(* IEC 61131-3 sources: brOscatLib/oscatNetw (part 2) *)

(* ---- DLOG_STORE_FILE_XML.st ---- *)
FUNCTION_BLOCK DLOG_STORE_FILE_XML
    (*http://www.oscat.de/images/OSCATBasic/oscat_basic333_en.pdf#page=46*)
    X.DTI := DTI; (* Datum / Zeit eintragen *)
    X.CLOCK_TRIG := DTI <> dti_last;
    dti_last := DTI;
    trig_auto := FALSE;
    IF X.CLOCK_TRIG THEN (* Impuls in jeder Sekunde *)
    	fn := DT_TO_STRF(DTI, 0, FILENAME, 0); (* automatische Dateinamen generierung *)
    	IF TRIG_T >= T#1000ms THEN (* automatischer Trigger *)
    		trig_auto := DT_TO_UDINT(DTI) MOD (TIME_TO_UDINT(TRIG_T) / UDINT#1000) = UDINT#0;
    	END_IF
    END_IF

    CASE step_1 OF

    00:	IF ENABLE THEN
    		aw_enable := AUTO_CLOSE >= T#5s;
    		wd_time := SEL(X.LOAD_TIME_MAX > T#0s, T#5ms,X.LOAD_TIME_MAX);
    		fn_last := fn; (* aktuellen Dateinnamen speichern *)
    		IF X.ID_MAX = USINT#0 THEN (* nur einmal nach Satellitenbausteinen scannen *)
    			X.ADD_COM := 01; (* ADD INFO *)
    			X.STORE_TYPE := BYTE#3; (* XML-Modus *)
    		END_IF
    		step_1 := 10;

    		(* ---------------- Debug-Message -----------------------*)
    		(*IF _debug_enable THEN
    			LOG_CL.NEW_MSG := 'FILE_XML1 - Start: File [~1], [~2]';
    			LOG_CL.PRINTF[1] := fn_last;
    			LOG_CL.PRINTF[2] := DT_TO_STRING(DTI);
    			LOG_MSG();
    		END_IF*)
    		(* -----------------------------------------------------------------*)

    	END_IF

    10:	X.UCB.D_STRING := fn_last;
    	IF fn_last = SAVE_DATA.FN_REM THEN
    		X.UCB.D_HEAD := WORD#16#F201; (* Filemode open + write *)
    		X.ADD_COM := 00;
    	ELSE
    		X.UCB.D_HEAD := WORD#16#F301; (* Filemode create + write *)
    		X.ADD_COM := 02; (* ADD HEADER *)
    	END_IF

    	X.UCB.D_MODE := 1; (* Dateinamen als String ablegen *)
    	UCB(DATA:=X.UCB); (* Daten eintragen *)
    	step_1 := 30;

    30:	(* LOG-Trigger verarbeiten *)
    	trig_tmp := (TRIG_M AND NOT trig_m_last) OR trig_auto OR X.ADD_DATA_REQ;

    	IF ENABLE = FALSE OR fn <> fn_last THEN (* ENABLE = 0 oder neuen Dateinamen -> Log Stop *)
    		trig_stored := trig_tmp; (* aktuellen Triggerpuls speichern *)
    		X.UCB.D_HEAD := WORD#16#EE00;
    		X.UCB.D_MODE := 1;
    		UCB(DATA:=X.UCB); (* Element schreiben *)
    		X.ADD_COM := 00;
    		step_1 := 00;

    		(* ---------------- Debug-Message -----------------------*)
    		(*IF _debug_enable THEN
    			LOG_CL.NEW_MSG := 'FILE_XML1 - Stop: [~2]';
    			LOG_CL.PRINTF[2] := DT_TO_STRING(DTI);
    			LOG_MSG();
    		END_IF*)
    		(* -----------------------------------------------------------------*)

    	ELSIF ENABLE THEN
    		IF trig_tmp OR trig_stored THEN (* manueller, automatischer oder externer Trigger *)
    			trig_stored := FALSE;
    			X.ADD_COM := 03; (* ADD DATA *)
    			SAVE_DATA.TRIG_CNT := SAVE_DATA.TRIG_CNT + UDINT#1;
    			SAVE_DATA.TRIG_CNT_TOTAL  := SAVE_DATA.TRIG_CNT_TOTAL + UDINT#1;
    			(* ---------------- Debug-Message -----------------------*)
    			(*IF _debug_enable THEN
    				LOG_CL.NEW_MSG := 'FILE_XML1 - Trig: [~2]';
    				LOG_CL.PRINTF[2] := DT_TO_STRING(DTI);
    				LOG_MSG();
    			END_IF*)
    			(* -----------------------------------------------------------------*)
    		ELSE
    			X.ADD_COM := 04;	(* ADD DATA REQ *)
    		END_IF
    	END_IF

    END_CASE
    X.ADD_DATA_REQ := FALSE; (* externe Anforderung rücksetzen *)

    (* ##################################### *)

    CASE step_2 OF

    00:	aw_ton(IN:= idx > 0 AND aw_enable , PT:= AUTO_CLOSE); (* AutoWrite Timer *)
    	IF aw_ton.Q THEN (* Zeitgesteuertes Datenschreiben *)
    		aw_aktiv := TRUE;
    		step_2 := 10; (* Daten schreiben *)
    		(* ---------------- Debug-Message -----------------------*)
    		(*IF _debug_enable THEN
    			LOG_CL.NEW_MSG := 'FILE_XML2 - AutoWrite: [~2]';
    			LOG_CL.PRINTF[2] := DT_TO_STRING(DTI);
    			LOG_MSG();
    		END_IF*)
    		(* -----------------------------------------------------------------*)

    	ELSE
    		wd_ton(IN:= FALSE, PT:= wd_time);
    		wd_ton(IN:= TRUE);
    		WHILE X.UCB.BUF_COUNT > 0 AND step_2 = 0 AND wd_ton.Q = FALSE DO

    			X.UCB.D_MODE := 10;
    			UCB(DATA:=X.UCB); (* Element lesen , aber noch nicht entfernen *)

    			IF X.UCB.D_HEAD > WORD#16#F000 THEN (* F301 oder F201 *)

    				str := '<?xml version="1.0" encoding="UTF-8"?><table>';

    				IF idx + LEN(str) < SIZEOF(PT.BUFFER) THEN (* Platz für Element vorhanden ? *)

    					FSD.MODE := WORD_TO_BYTE(SHR(SHL(X.UCB.D_HEAD,4),12)); (* 0X00 -> 000X = 3 create + write / 2 open + write *)
    					FSD.OFFSET := UDINT#0; (* Start bei Dateianfang *)
    					FSD.FILENAME := X.UCB.D_STRING; (* Dateiname *)
    					PT.SIZE := UINT#0;
    					SAVE_DATA.FN_REM := FSD.FILENAME; (* aktuellen Dateinamen remanent sichern *)

    					X.NEW_FILE := FSD.FILENAME;
    					X.NEW_FILE_SIZE := UDINT#0;
    					X.NEW_FILE_RTRIG := FALSE;
    					step_2 := 20;

    					(* Headerdaten schreiben *)
    					IF FSD.MODE = BYTE#3 THEN
    						SAVE_DATA.TRIG_CNT := UDINT#0; (* Datei neu anlegen -> dann zähler reset *)

    						_STRING_TO_BUFFER(str:=str, POS:=idx, PT:=ADR(PT.BUFFER), SIZE:=SIZEOF(PT.BUFFER));
    						idx := idx + LEN(str);
    						X.NEW_FILE_SIZE := total_bytes + INT_TO_UDINT(idx);
    					END_IF

    					X.UCB.D_MODE := 11;
    					UCB(DATA:=X.UCB); (* Element entfernen *)

    					(* ---------------- Debug-Message -----------------------*)
    					(*IF _debug_enable THEN
    						LOG_CL.NEW_MSG := 'FILE_XML2 - Create: Mode [~1] , [~2]';
    						LOG_CL.PRINTF[2] := DT_TO_STRING(DTI);
    						LOG_CL.PRINTF[1] := BYTE_TO_STRING(FSD.MODE);
    						LOG_MSG();
    					END_IF*)
    					(* -----------------------------------------------------------------*)
    				END_IF

    			ELSIF X.UCB.D_HEAD = WORD#16#EE00 THEN (* log_stop Command *)

    				str := '</table>';

    				IF idx + LEN(str) < SIZEOF(PT.BUFFER) THEN (* Platz für Element vorhanden ? *)

    					_STRING_TO_BUFFER(str:=str, POS:=idx, PT:=ADR(PT.BUFFER), SIZE:=SIZEOF(PT.BUFFER));
    					idx := idx + LEN(str);
    					log_stop := TRUE;
    					step_2 := 10; (* Daten schreiben *)

    					X.UCB.D_MODE := 11;
    					UCB(DATA:=X.UCB); (* Element entfernen *)

    				END_IF

    			ELSIF idx + LEN(X.UCB.D_STRING) + 120 < SIZEOF(PT.BUFFER) THEN (* Platz für Element vorhanden ? *)

    				(* ---------------- Debug-Message -----------------------*)
    				(*IF _debug_enable THEN
    					LOG_CL.NEW_MSG := 'FILE_XML2 - BUF: TXT [~1],Pos [~2], [~3]';
    					LOG_CL.PRINTF[1] := X.UCB.D_STRING;
    					LOG_CL.PRINTF[2] := INT_TO_STRING(idx);
    					LOG_CL.PRINTF[3] := DT_TO_STRING(DTI);
    					LOG_MSG();
    				END_IF*)
    				(* -----------------------------------------------------------------*)

    				IF log_state = USINT#0 THEN
    					str := '<row><entry>';
    				ELSE
    					str := '<entry>';
    				END_IF

    				_STRING_TO_BUFFER(str:=str, POS:=idx, PT:=ADR(PT.BUFFER), SIZE:=SIZEOF(PT.BUFFER));
    				idx := idx + LEN(str);
    				log_state := log_state + USINT#1;

    				_STRING_TO_BUFFER(str:=X.UCB.D_STRING, POS:=idx, PT:=ADR(PT.BUFFER), SIZE:=SIZEOF(PT.BUFFER));
    				idx := idx + LEN(X.UCB.D_STRING);

    				n := n + USINT#1;
    				IF n >= X.ID_MAX THEN
    					n := USINT#0;
    					str := '</entry></row>';
    					log_state := USINT#0;
    				ELSE
    					str := '</entry>';
    				END_IF
    				_STRING_TO_BUFFER(str:=str, POS:=idx, PT:=ADR(PT.BUFFER), SIZE:=SIZEOF(PT.BUFFER));
    				idx := idx + LEN(str);
    				X.NEW_FILE_SIZE := total_bytes + INT_TO_UDINT(idx);

    				X.UCB.D_MODE := 11;
    				UCB(DATA:=X.UCB); (* Element entfernen *)

    			ELSE (* kein Platz vorhanden *)
    				step_2 := 10; (* Daten schreiben *)
    			END_IF
    			wd_ton();
    		END_WHILE
    	END_IF

    10:	IF idx > 0 THEN (* Daten schreiben *)
    		FSD.MODE := BYTE#2; (* File_Open_Exist + File_Write *)
    		FSD.OFFSET := UDINT#4294967294; (* 16#FFFF_FFFE ->Spezialcode: Daten automatisch an Dateiende anhängen *)
    		PT.SIZE := INT_TO_UINT(idx); (* Datenlänge eintragen *)
    		idx := 0;
    		(* ---------------- Debug-Message -----------------------*)
    		(*IF _debug_enable THEN
    			LOG_CL.NEW_MSG := 'FILE_XML2 - WriteData: Mode [~3] Size [~1] , [~2]';
    			LOG_CL.PRINTF[1] := UINT_TO_STRING(PT.SIZE);
    			LOG_CL.PRINTF[2] := DT_TO_STRING(DTI);
    			LOG_CL.PRINTF[3] := BYTE_TO_STRING(FSD.MODE);
    			LOG_MSG();
    		END_IF*)
    		(* -----------------------------------------------------------------*)
    	END_IF
    	step_2 := 20;

    20:	IF FSD.MODE = BYTE#0 THEN
    		total_bytes := FSD.FILE_SIZE;
    		X.NEW_FILE_SIZE := total_bytes + INT_TO_UDINT(idx);
    		IF log_stop OR aw_aktiv THEN
    			aw_aktiv := FALSE;
    			FSD.MODE := BYTE#5; (* Datei schliessen *)
    			(* ---------------- Debug-Message -----------------------*)
    			(*IF _debug_enable THEN
    				LOG_CL.NEW_MSG := 'FILE_XML2 - Close: [~2]';
    				LOG_CL.PRINTF[2] := DT_TO_STRING(DTI);
    				LOG_MSG();
    			END_IF*)
    			(* -----------------------------------------------------------------*)
    		END_IF
    		step_2 := 30;
    	END_IF

    30:	IF FSD.MODE = BYTE#0 THEN (* Datei schliessen beendet *)
    		IF log_stop THEN
    			X.NEW_FILE_RTRIG := TRUE;
    			log_stop := FALSE;
    			SAVE_DATA.FN_REM := ''; (* remanenten Dateinamen löschen *)
    		END_IF
    		step_2 := 00;
    	END_IF

    END_CASE

    FS(FSD:=FSD,PT:=PT); (* FILE_SERVER *)

    (* Fehlerauswertung *)
    IF FSD.ERROR <> BYTE#0 THEN
    	ERROR_C := BYTE_TO_DWORD(FSD.ERROR);
    	ERROR_T := BYTE#1;
    ELSIF X.UCB.BUF_DATA_LOST > UDINT#0 THEN
    	ERROR_C := DWORD#2; (* Fehler: Bufferüberlauf - Datenmenge reduzieren *)
    	ERROR_T := BYTE#6; 	(* Type: Buffer *)
    ELSIF X.UCB.BUF_USED_MAX > USINT#90 THEN
    	ERROR_C := DWORD#1; (* Warnung: Buffer auslastung > 90% *)
    	ERROR_T := BYTE#6;	(* Type: Buffer *)
    ELSE
    	ERROR_C := DWORD#0;
    	ERROR_T := BYTE#0;
    END_IF

    trig_m_last := TRIG_M;

    (* revision history
    ks	25. july. 2011	rev 1.0
    	original version

    ks	16. apr. 2012	rev 1.1
    	neuer überarbeiteter Code für automatisches File-open/close

    ks	8. mar. 2016	rev 1.2
    	nur einmal nach satellitenbausteinen scannen

    ks	21. mar. 2016	rev 1.3
    	prüfung auf freien bufferplatz hinzugefügt
    	fehlermeldungen hinzugefügt

    *)
END_FUNCTION_BLOCK

(* ---- DLOG_STORE_MYSQL.st ---- *)
FUNCTION_BLOCK DLOG_STORE_MYSQL
    (*http://www.oscat.de/images/OSCATBasic/oscat_basic333_en.pdf#page=46*)
    X.DTI := DTI; (* Datum / Zeit eintragen *)
    X.CLOCK_TRIG := DTI <> dti_last;
    dti_last := DTI;
    trig_auto := FALSE;
    IF X.CLOCK_TRIG THEN (* Impuls in jeder Sekunde *)
    	del_start := DT_TO_UDINT(DTI) - del_dt > AUTO_DELETE AND AUTO_DELETE > UDINT#0;
    	IF TRIG_T >= T#1000ms THEN (* automatischer Trigger *)
    		trig_auto := DT_TO_UDINT(DTI) MOD (TIME_TO_UDINT(TRIG_T) / UDINT#1000) = UDINT#0;
    	END_IF
    END_IF
    X.ADD_COM := 00;

    CASE step OF

    00:	IF ENABLE AND enable_last = FALSE THEN
    		y.SQL_URL := URL;
    		y.TIMEOUT := TIMEOUT;
    		y.DNS_IP4 := DNS_IP4;
    		y.SQL_CON := TRUE;

    		X.UCB.D_MODE := 99; (* Buffer reset - Alles löschen *)
    		UCB(DATA:=X.UCB);

    		IF X.ID_MAX = USINT#0 THEN (* nur einmal nach Satellitenbausteinen scannen *)
    			X.ADD_COM := 01; (* ADD INFO *)
    			X.STORE_TYPE := BYTE#5; (* MySQL-Modus *)
    		END_IF

    		step := 05;
    	END_IF

    05:	X.ADD_COM := 02; (* ADD HEADER *)
    	step := 10;

    10:	IF SQL_INFO.SQL_CONNECTED THEN
    		sql_command := BYTE#3; (* CREATE DATABASE IF NOT EXISTS `DB_NAME` *)
    		snd_text :=  CONCAT('CREATE DATABASE IF NOT EXISTS `' ,DB_NAME);
    		snd_text :=  CONCAT(snd_text, '`');
    		next_step := 20;
    	END_IF

    20:	sql_command := BYTE#2; (* 0x02 COM_INIT_DB mysql_select_db *)
    	snd_text := DB_NAME;
    	next_step := 30;

    30:	(* CREATE TABLE IF NOT EXISTS TB_NAME (Timestamp TIMESTAMP NULL DEFAULT CURRENT_TIMESTAMP, n1,n2) *)
    	sql_command := BYTE#0;
    	idx := 5;
    	n := USINT#0;
    	WHILE sql_command = BYTE#0 DO
    		IF n = USINT#0 THEN
    			snd_text := CONCAT('CREATE TABLE IF NOT EXISTS `', TB_NAME);
    			snd_text := CONCAT(snd_text,'` (`ID` BIGINT NOT NULL AUTO_INCREMENT PRIMARY KEY ,');
    			snd_text := CONCAT(snd_text,' store_timestamp TIMESTAMP NULL DEFAULT CURRENT_TIMESTAMP');
    		ELSIF n <= X.ID_MAX THEN
    			X.UCB.D_MODE := 12; (* Element lesen und löschen *)
    			UCB(DATA:=X.UCB);
    			snd_text := CONCAT(', `',X.UCB.D_STRING);
    			CASE WORD_TO_INT(SHR(X.UCB.D_HEAD,8)) OF
    			02:	snd_text := CONCAT(snd_text, '` FLOAT'); (* REAL *)
    			06:	snd_text := CONCAT(snd_text, '` BOOL'); (* BOOL *)
    			08:	snd_text := CONCAT(snd_text, '` INT'); (* DINT *)
    			13:	snd_text := CONCAT(snd_text, '` DATETIME'); (* DT *)
    			ELSE
    				snd_text := CONCAT(snd_text, '` VARCHAR(80)'); (* STRING(80) *)
    			END_CASE
    		ELSE
    			snd_text := ')';
    			sql_command := BYTE#3;
    			snd_size := idx + LEN(snd_text);
    			next_step := 40;
    		END_IF
    		_STRING_TO_BUFFER(str:=snd_text,pos:=idx,pt:=ADR(y.S_BUF.BUFFER),size:=SIZEOF(y.S_BUF.BUFFER)); (* String in puffer kopieren *)
    		idx := idx + LEN(snd_text);
    		n := n + USINT#1;

    		(*####################  DEBUG-MESSAGE  ###################################*)
    		(*IF _debug_enable THEN
    			LOG_CL.NEW_MSG := 'dlog_mysql: create >~1<';
    			LOG_CL.PRINTF[1] := snd_text;
    			LOG_MSG();
    		END_IF*)
    		(*########################################################################*)
    	END_WHILE

    40:	IF del_start THEN
    		del_start := FALSE;
    		sql_command := BYTE#3; (* DELETE FROM `TB_NAME` WHERE TIMESTAMPDIFF(SECOND, Timestamp, NOW()) > xxx *)
    		snd_text := CONCAT('DELETE FROM `', TB_NAME);
    		snd_text := CONCAT(snd_text, '` WHERE TIMESTAMPDIFF(SECOND, store_timestamp, NOW()) > ');
    		snd_text := CONCAT(snd_text, UDINT_TO_STRING(AUTO_DELETE));
    		next_step := 40;
    		del_dt := DT_TO_UDINT(DTI);
    		(*####################  DEBUG-MESSAGE  ###################################*)
    		(*IF _debug_enable THEN
    			LOG_CL.NEW_MSG := 'dlog_mysql: # delete time:~1 >~2<';
    			LOG_CL.PRINTF[1] := UDINT_TO_STRING(AUTO_DELETE);
    			LOG_CL.PRINTF[2] := snd_text;
    			LOG_MSG();
    		END_IF*)
    		(*########################################################################*)

             (* INSERT INTO `TB_NAME` VALUES (CURRENT_TIMESTAMP,  "n1","n2") *)
    	ELSIF X.UCB.BUF_COUNT >= USINT_TO_INT(X.ID_MAX) AND step > 0 THEN (* Neue Datenreihe(n) vorhanden *)
    		idx := 5;
    		n := USINT#0;
    		sql_command := BYTE#0;
    		WHILE sql_command = BYTE#0 DO
    			IF n = USINT#0 THEN
    				snd_text := CONCAT('INSERT INTO `', TB_NAME);
    				snd_text := CONCAT(snd_text,'` VALUES (NULL, CURRENT_TIMESTAMP');
    			ELSIF n <= X.ID_MAX THEN
    				X.UCB.D_MODE := 12; (* Element lesen und löschen *)
    				UCB(DATA:=X.UCB);
    				snd_text := CONCAT(', "',X.UCB.D_STRING);
    				snd_text := CONCAT(snd_text, '"');
    			ELSE
    				snd_text := ')';
    				sql_command := BYTE#3;
    				snd_size := idx + LEN(snd_text);
    				next_step := 40;
    			END_IF
    			_STRING_TO_BUFFER(str:=snd_text,pos:=idx,pt:=ADR(y.S_BUF.BUFFER),size:=SIZEOF(y.S_BUF.BUFFER)); (* String in puffer kopieren *)
    			idx := idx + LEN(snd_text);
    			n := n + USINT#1;

    			(*####################  DEBUG-MESSAGE  ###################################*)
    			(*IF _debug_enable THEN
    				LOG_CL.NEW_MSG := 'dlog_mysql: insert >~1<';
    				LOG_CL.PRINTF[1] := snd_text;
    				LOG_MSG();
    			END_IF*)
    			(*########################################################################*)
    		END_WHILE
    	END_IF

    	IF ENABLE THEN 	(* LOG-Trigger verarbeiten *)
    		trig_tmp := (TRIG_M AND NOT trig_m_last) OR trig_auto OR X.ADD_DATA_REQ;

    		IF trig_tmp THEN (* manueller, automatischer oder externer Trigger *)
    			X.ADD_COM := 03; (* ADD DATA *)
    			(* ---------------- Debug-Message -----------------------*)
    			(*IF _debug_enable THEN
    				LOG_CL.NEW_MSG := 'dlog_mysql: Trigger: DATE [~2]';
    				LOG_CL.PRINTF[2] := DT_TO_STRING(DTI);
    				LOG_MSG();
    			END_IF*)
    			(* -----------------------------------------------------------------*)
    		ELSE
    			X.ADD_COM := 04;	(* ADD DATA REQ *)
    		END_IF
    	ELSE
    		y.SQL_CON := FALSE; (* MySQL Verbindung beenden *)
    		step := 0;
    	END_IF
    	X.ADD_DATA_REQ := FALSE;

    (* ~~~~~~~~~~~~~~~~~~~~~~ *)

    199:IF y.SQL_RCV_STATE = BYTE#1 THEN (* OK *)
    		step := next_step;
    	ELSIF y.SQL_RCV_STATE = BYTE#2 THEN  (* FEHLER *)
    		step := 0;
    	END_IF

    END_CASE

    (* ########################## *)
    (* SQL-Kommando ausführen *)
    IF sql_command > BYTE#0 THEN

    	IF snd_size > 0 THEN
    		y.S_BUF.SIZE := INT_TO_UINT(snd_size);
    		snd_size := 0;
    	ELSE
    		_STRING_TO_BUFFER(str:=snd_text,pos:=5,pt:=ADR(y.S_BUF.BUFFER),size:=SIZEOF(y.S_BUF.BUFFER)); (* String in puffer kopieren *)
    		y.S_BUF.SIZE := INT_TO_UINT(5 + LEN(snd_text));
    		snd_text := '';
    	END_IF

    	IF y.S_BUF.SIZE > SIZEOF(y.S_BUF.BUFFER) THEN (* buffer überlauf erkannt -> Abbruch *)
    		y.S_BUF.SIZE := 0;
    		sql_command := BYTE#0;
    		y.SQL_CON := FALSE; (* MySQL Verbindung beenden *)
    		step := 999; (* Dummy-Schritt *)
    	ELSE

    		i2 := UINT_TO_INT(y.S_BUF.SIZE) - 1; (* alle " zeichen mit ' ersetzen *)
    		FOR i1 := 5 TO i2 DO
    			IF y.S_BUF.BUFFER[i1] = BYTE#34 THEN
    				y.S_BUF.BUFFER[i1] := BYTE#39;
    			END_IF
    		END_FOR

    		y.S_BUF.BUFFER[4] := sql_command;
    		y.SQL_PACKET_NO := BYTE#255;
    		sql_command := BYTE#0;
    		step := 199;
    	END_IF
    END_IF

    (* ########################## *)

    MYSQL_CONTROL(COM:= y, INFO:=SQL_INFO);

    (* Fehlerauswertung *)
    IF step = 999 THEN	(* Buffer überlauf *)
    	ERROR_C := DWORD#3; (* Netzwerkbuffer überlauf *)
    	ERROR_T := BYTE#6; 	(* Type: Buffer *)
    ELSIF y.ERROR_T > BYTE#0 THEN	(* SQL Error *)
    	ERROR_C := y.ERROR_C;
    	ERROR_T := y.ERROR_T;
    	step := 0;
    ELSIF X.UCB.BUF_DATA_LOST > UDINT#0 THEN
    	ERROR_C := DWORD#2; (* Fehler: Bufferüberlauf - Datenmenge reduzieren *)
    	ERROR_T := BYTE#6; 	(* Type: Buffer *)
    ELSIF X.UCB.BUF_USED_MAX > USINT#90 THEN
    	ERROR_C := DWORD#1; (* Warnung: Buffer auslastung > 90% *)
    	ERROR_T := BYTE#6;	(* Type: Buffer *)
    ELSE
    	ERROR_C := DWORD#0;
    	ERROR_T := BYTE#0;
    END_IF

    (* ########################## *)

    trig_m_last := TRIG_M;
    enable_last := ENABLE;
    run := step > 0;

    (* revision history
    ks	20. apr. 2012	rev 1.0
    	original version

    ks	17. jan. 2014	rev 1.1
    	DELTA Error

    ks	8. mar. 2016	rev 1.2
    	nur einmal nach satellitenbausteinen scannen

    ks	21. mar. 2016	rev 1.3
    	prüfung auf bufferüberlauf und fehlermeldungen hinzugefügt

    *)
END_FUNCTION_BLOCK

(* ---- DLOG_STORE_RRD.st ---- *)
FUNCTION_BLOCK DLOG_STORE_RRD
    (*http://www.oscat.de/images/OSCATNetwork/oscat_netlib121_en.pdf#page=54*)
    X.DTI := DTI; (* Datum / Zeit eintragen *)
    X.CLOCK_TRIG := DTI <> dti_last;
    dti_last := DTI;
    trig_auto := FALSE;
    IF X.CLOCK_TRIG THEN (* Impuls in jeder Sekunde *)
    	IF TRIG_T >= T#1000ms THEN (* automatischer Trigger *)
    		trig_auto := DT_TO_UDINT(DTI) MOD (TIME_TO_UDINT(TRIG_T) / UDINT#1000) = UDINT#0;
    	END_IF
    END_IF

    CASE step_1 OF

    00:	IF ENABLE THEN
    		IF X.ID_MAX = USINT#0 THEN (* nur einmal nach Satellitenbausteinen scannen *)
    			X.ADD_COM := 01; (* ADD INFO *)
    			X.STORE_TYPE := BYTE#1; (* RRD-Modus *)
    		END_IF

    		ERROR_T := BYTE#0;
    		ERROR_C := DWORD#0;

    		X.UCB.D_MODE := 99;
    		UCB(DATA:=X.UCB); (* Buffer löschen *)

    		URL_DATA:=STRING_TO_URL(STR:=URL,DEFAULT_PROTOCOL:='',DEFAULT_PATH:=''); (* URL zerlegen *)
    		sep_char := CHR_TO_STRING(SEP);
    		url_query := URL_DATA.QUERY;
    		step_1 := 30;

    		(* ---------------- Debug-Message -----------------------*)
    		(*IF _debug_enable THEN
    			LOG_CL.NEW_MSG := 'FILE_RRD1 - Start: DATE [~2]';
    			LOG_CL.PRINTF[2] := DT_TO_STRING(DTI);
    			LOG_MSG();
    		END_IF*)
    		(* -----------------------------------------------------------------*)

    	END_IF

    30:	(* LOG-Trigger verarbeiten *)
    	trig_tmp := (TRIG_M AND NOT trig_m_last) OR trig_auto OR X.ADD_DATA_REQ;

    	IF ENABLE = FALSE THEN (* ENABLE = 0 -> Log Stop *)
    		X.ADD_COM := 00;
    		step_1 := 00;

    		(* ---------------- Debug-Message -----------------------*)
    		(*IF _debug_enable THEN
    			LOG_CL.NEW_MSG := 'FILE_RRD1 - Stop: DATE [~2]';
    			LOG_CL.PRINTF[2] := DT_TO_STRING(DTI);
    			LOG_MSG();
    		END_IF*)
    		(* -----------------------------------------------------------------*)

    	ELSIF ENABLE THEN
    		IF trig_tmp OR trig_stored THEN (* manueller, automatischer oder externer Trigger *)
    			trig_stored := FALSE;
    			X.ADD_COM := 03; (* ADD DATA *)
    			(* ---------------- Debug-Message -----------------------*)
    			(*IF _debug_enable THEN
    				LOG_CL.NEW_MSG := 'FILE_RRD1 - Trig: DATE [~2]';
    				LOG_CL.PRINTF[2] := DT_TO_STRING(DTI);
    				LOG_MSG();
    			END_IF*)
    			(* -----------------------------------------------------------------*)
    		ELSE
    			X.ADD_COM := 04;	(* ADD DATA REQ *)
    		END_IF
    	END_IF

    END_CASE
    X.ADD_DATA_REQ := FALSE; (* externe Anforderung rücksetzen *)

    (* ##################################### *)

    CASE step_2 OF

    00:	IF X.UCB.BUF_DATA_LOST > UDINT#0 THEN
    		ERROR_C := DWORD#2; (* Fehler: Bufferüberlauf - Datenmenge reduzieren *)
    		ERROR_T := BYTE#6; 	(* Type: Buffer *)
    		step_2 := 100;
    	ELSIF X.UCB.BUF_USED_MAX > USINT#90 THEN
    		ERROR_C := DWORD#1; (* Warnung: Buffer auslastung > 90% *)
    		ERROR_T := BYTE#6;	(* Type: Buffer *)
    	END_IF

    	IF X.UCB.BUF_COUNT >= USINT_TO_INT(X.ID_MAX) THEN (* genug Einträge vorhanden *)
    		URL_DATA.QUERY := url_query; (* original Query wiederherstellen *)
    		n := 1;
    		WHILE n <= USINT_TO_INT(X.ID_MAX) DO
    			X.UCB.D_MODE := 12; (* Element lesen und löschen *)
    			UCB(DATA:=X.UCB);
    			IF n < USINT_TO_INT(X.ID_MAX) THEN (* Trennzeichen hinzufügen *)
    				X.UCB.D_STRING := CONCAT(X.UCB.D_STRING,sep_char);
    			END_IF
    			IF LEN(X.UCB.D_STRING) + LEN(URL_DATA.QUERY) <= STRING_LENGTH THEN
    				URL_DATA.QUERY := CONCAT(URL_DATA.QUERY,X.UCB.D_STRING); (* Query mit LOG-Daten ergänzen *)
    				step_2 := 40;
    			ELSE
    				ERROR_T := BYTE#4; (* LOG-Daten können nicht in URL gepackt werden *)
    				ERROR_C := DWORD#1;
    				step_2 := 100;
    			END_IF
    			n := n + 1;
    		END_WHILE;
    	END_IF

    40:	IF DNS_CLIENT.DONE THEN
    		step_2 := 60;
    	ELSIF (DNS_CLIENT.ERROR > DWORD#0) THEN
    		ERROR_C := DNS_CLIENT.ERROR; (* Fehlerbehandlung *)
    		ERROR_T := BYTE#1;
    		step_2 := 100;
    	END_IF

    60:	IF HTTP_GET.DONE THEN
    		n := UINT_TO_INT(HTTP_GET.BODY_START);
    		IF R_BUF.BUFFER[n] <> BYTE#48 THEN (* ASCII '0' *)
    			ERROR_C := DWORD#1;
    			ERROR_T := BYTE#3;
    		END_IF
    		step_2 := 100;

    	ELSIF HTTP_GET.ERROR > DWORD#0 THEN (* Fehlerbehandlung *)
    		ERROR_C := HTTP_GET.ERROR;
    		ERROR_T := BYTE#2;
    		step_2 := 100;
    	END_IF

    100:	IF (NOT HTTP_GET.DONE) THEN (* UNLOCK HTTP DATA *)
    		step_2 := SEL(ERROR_T = BYTE#0, 120,0);
    	END_IF

    120:	IF NOT ENABLE THEN
    		step_2 := 0;
    	END_IF

    END_CASE

    HTTP_GET(IP_C:=IP_C,S_BUF:=S_BUF,R_BUF:=R_BUF,IP4:=DNS_CLIENT.IP4,GET:=step_2=60,MODE:=2,UNLOCK_BUF:=step_2=100,URL_DATA:=URL_DATA); (* HTTP_GET *)
    DNS_CLIENT(IP_C:=IP_C, S_BUF:=S_BUF, R_BUF:=R_BUF, DOMAIN:=URL_DATA.DOMAIN, IP4_DNS:= DNS_IP4, ACTIVATE:=step_2=40); (* DNS-Client *)
    IPC(IP:= 0, PORT:= 0 , TIME_OUT:= TIMEOUT, IP_C:= IP_C, S_BUF:= S_BUF, R_BUF:= R_BUF); (* IP_CONTROL *)

    trig_m_last := TRIG_M;

    (* revision history
    ks	01. jan. 2011	rev 1.0
    	original version

    ks	13. may. 2011	rev 1.1
    	ADD_DATA_REQ hinzugefügt

    ks	26. july. 2011	rev 1.2
    	code optimierung D_MODE 12 und bessere fehlerauswertung

    ks	16. apr. 2012	rev 1.3
    	neuer überarbeiteter Code

    ks	21. mar. 2016	rev 1.4
    	nur einmal nach satellitenbausteinen scannen und fehlermeldungen hinzugefügt

    *)
END_FUNCTION_BLOCK

(* ---- DLOG_STRING.st ---- *)
FUNCTION_BLOCK DLOG_STRING
    (*http://www.oscat.de/images/OSCATNetwork/oscat_netlib121_en.pdf#page=52*)
    CASE X.ADD_COM OF

    01:	(* ADD INFO *)
    	X.ID_MAX := X.ID_MAX + USINT#1;
    	id := WORD#16#0101; (* Quelltype STRING , Zieltype STRING *)
    02:	(* ADD HEADER *)
    	X.UCB.D_STRING := COLUMN;
    	X.UCB.D_HEAD := id;
    	X.UCB.D_MODE := 1;
    	UCB(DATA:=X.UCB); (* Daten eintragen *)
    03:	(* ADD DATA *)
    	X.UCB.D_STRING := str_last;
    	X.UCB.D_HEAD := id;
    	X.UCB.D_MODE := 1;
    	UCB(DATA:=X.UCB); (* Daten eintragen *)
    END_CASE
    str_last := STR;

    (* revision history
    ks	01. jan. 2011	rev 1.0
    	original version

    ks	17. may. 2011	rev 1.1
    	COLUMN STRING(40)

    ks	25. july.   2011	rev 1.2
    	neue head information

    ks	19. apr.   2012	rev 1.3
    	code neu überarbeitet
    *)
END_FUNCTION_BLOCK

(* ---- DNS_CLIENT.st ---- *)
FUNCTION_BLOCK DNS_CLIENT
    (*http://www.oscat.de/images/OSCATNetwork/oscat_netlib121_en.pdf#page=89*)
    (* DOMAIN Name System (query) *)

    CASE state OF

    00:	IF ACTIVATE AND NOT activate_last THEN (* auf positive Flanke GET warten *)
    		DONE := FALSE;
    		ERROR := DWORD#0;
    		state := 5;
    	END_IF

    05:	IP4 := IP4_DECODE(str:=DOMAIN); (* prüfe ob DOMAIN schon eine IP4-Adresse ist *)
    	IF IP4 > DWORD#00 THEN
    		DONE := TRUE;
    		state := 0;
            		(*####################  DEBUG-MESSAGE  ###################################*)
            		(*IF _debug_enable THEN
                		LOG_CL.NEW_MSG := 'DNS: S05 IP4 ~1';
                		LOG_CL.PRINTF[1]  := DOMAIN;
                		LOG_MSG();
            		END_IF*)
            		(*########################################################################*)
    	ELSE
    		ip_state := BYTE#1;
    		ttl_last := DWORD#0;
    		domain_copy := DOMAIN; (* DOMAIN String sichern *)
    		state := 10;
            		(*####################  DEBUG-MESSAGE  ###################################*)
            		(*IF _debug_enable THEN
                		LOG_CL.NEW_MSG := 'DNS: S05 START';
                		LOG_MSG();
            		END_IF*)
            		(*########################################################################*)
    	END_IF

    10:	IF ip_state = BYTE#3 THEN (* Bei IP_Control anmelden *)
    		url_length := LEN(domain_copy);
    		char_count := 17 + url_length; (* sendebuffer initialisieren *)
    		FOR i := 0 TO char_count DO
    			S_BUF.BUFFER[i] := BYTE#00;
    		END_FOR
    		tid := UINT_TO_BYTE(BYTE_TO_UINT(tid) + UINT#1);
    		S_BUF.BUFFER[01] := tid; (* Transaction ID lowbyte *)
    		S_BUF.BUFFER[02] := BYTE#16#01; (* Flags: highbyte *)
    		S_BUF.BUFFER[05] := BYTE#16#01; (* Questions: lowbyte *)
    		i := url_length + 12;	(* den servernamen von hinten nach vorne bearbeiten *)
    		char_count := 0;
    		WHILE i > 12 DO
    			char := CODE(STR:=domain_copy,POS:=i - 12);
    			IF char = BYTE#46 THEN (* prüfe auf haupt/sub domänen namens-teiler "." *)
    				S_BUF.BUFFER[i] := INT_TO_BYTE(char_count); (* anstelle des teilers "." wird die länge des erkannten haupt/sub domänennames eingetragen *)
    				char_count := 0;
    			ELSE
    				S_BUF.BUFFER[i] := char; (* char in buffer eintragen *)
    				char_count := char_count + 1; (* anzahl char zählen *)
    			END_IF
    			i := i - 1;
    		END_WHILE
    		S_BUF.BUFFER[i] := INT_TO_BYTE(char_count); (* längenangabe des ganz linken (ersten) domänennamens eintragen *)
    		i := url_length + 15; (* position hinter dem servernamen *)
    		S_BUF.BUFFER[i] := BYTE#01; (* Type: A Hostaddress lowbyte *)
    		i := i + 2;
    		S_BUF.BUFFER[i] := BYTE#01; (* Class: IN lowbyte *)
    		i := i + 1;
    		(* IP Datenverkehr einrichten *)
    		IP_C.C_PORT := WORD#53; (* Portnummer eintragen *)
    		IP_C.C_IP := IP4_DNS; (* IP eintragen *)
    		IP_C.C_MODE := BYTE#1; (* Mode: UDP+AKTIV+PORT+IP *)
    		IP_C.C_ENABLE := TRUE; (* Verbindungsaufbau freigeben *)
    		IP_C.TIME_RESET := TRUE; (* Zeitueberwachung rücksetzen *)
    		IP_C.R_OBSERVE  := TRUE; (* Datenempfang ueberwachen *)
    		S_BUF.SIZE := INT_TO_UINT(i); (* sendelänge eintragen *)
    		R_BUF.SIZE := UINT#0; (* Empfangslänge rücksetzen *)
    		state := 30;

            		(*####################  DEBUG-MESSAGE  ###################################*)
            		(*IF _debug_enable THEN
                		LOG_CL.NEW_MSG := 'DNS: S10 SEND';
                		LOG_MSG();
            		END_IF*)
            		(*########################################################################*)
    	END_IF

    30:	IF IP_C.ERROR <> DWORD#00 THEN
    		ERROR := IP_C.ERROR;
    		state := 99;
            		(*####################  DEBUG-MESSAGE  ###################################*)
            		(*IF _debug_enable THEN
                		LOG_CL.NEW_MSG := 'DNS: S30 ERROR ~1';
                		LOG_CL.PRINTF[1]  := DWORD_TO_STRING(ERROR);
                		LOG_MSG();
            		END_IF*)
            		(*########################################################################*)

    	ELSIF (S_BUF.SIZE = UINT#0) AND (tid = R_BUF.BUFFER[1]) AND (R_BUF.SIZE >= INT_TO_UINT(34 + url_length)) THEN	(* prüfe ob antwort telegramm die richtige Transaction-ID und mindestlänge hat *)
    		ERROR := BYTE_TO_DWORD(R_BUF.BUFFER[3] AND BYTE#2#0000_1111); (* prüfe Return code der Flags. 4 bits *)
    		IF ERROR = DWORD#00 THEN
    			anc := R_BUF.BUFFER[7]; (* Anzahl der Answer-RR *)
    			IP_C.R_OBSERVE := FALSE; (* Datenempfang ueberwachen *)
    			state := 40;
    		ELSE
    			state := 99;
    		END_IF
    	END_IF

    40:	IF anc > 0 THEN
    		anc := anc - 1;
    		WHILE i < R_BUF.SIZE DO
    			x := R_BUF.BUFFER[i];
    			IF rr_stop = FALSE THEN
    				IF x > BYTE#63 THEN (* zeiger auf namen *)
    					i := i + 1;
    					rr_stop := TRUE;
    				ELSIF x= BYTE#0 THEN (* namens ende *)
    					rr_stop := TRUE;
    				ELSE
    					i := i + x; (* namen *)
    				END_IF
    				i := i + 1;
    			ELSE
    				rr_stop := FALSE;
    				IF R_BUF.BUFFER[i+1] = BYTE#1 AND R_BUF.BUFFER[i+3] = BYTE#1 THEN (* Type A / Class IN *)
    					i := i + 4;
    					ttl_tmp := DWORD_OF_BYTE(R_BUF.BUFFER[i],R_BUF.BUFFER[i+1],R_BUF.BUFFER[i+2],R_BUF.BUFFER[i+3]); (* Time to live *)
    					i := i + 6;
    					IF ttl_tmp >= ttl_last THEN (* TTL ist länger *)
    						ttl_last := ttl_tmp;
    						IP4 := DWORD_OF_BYTE(R_BUF.BUFFER[i],R_BUF.BUFFER[i+1],R_BUF.BUFFER[i+2],R_BUF.BUFFER[i+3]); (* IP-Adresse *)
    					END_IF
    					i := i + 4;
    				ELSE
    					i := i + 9;
    					i := i + R_BUF.BUFFER[i] + 1; (* offset zu nächsten Block *)
    				END_IF
    				EXIT;
    			END_IF
    		END_WHILE
    	ELSE
    		IF IP4 > DWORD#0 THEN (* gültige RR mit IP gefunden *)
    			DONE := TRUE;
                		(*####################  DEBUG-MESSAGE  ###################################*)
                		(*IF _debug_enable THEN
                    			LOG_CL.NEW_MSG := 'DNS: S40 OK';
                    			LOG_MSG();
                		END_IF*)
                		(*########################################################################*)
    		ELSE
    			ERROR := DWORD#255; (* Daten fehlerhaft - keine IP-Adresse vorhanden *)
    		END_IF
    		state := 99;
    	END_IF

    99:	R_BUF.SIZE := UINT#0; (* Empfangslänge rücksetzen *)
    	ip_state := BYTE#4; (* Abmelden *)
    	state := 00;

    END_CASE

    activate_last := ACTIVATE; (* letzten Status sichern zur Flankenerkennung *)
    IP_FIFO(FIFO:=IP_C.FIFO,state:=ip_state,ID:=ip_id); (* IP_FIFO *)

    (* revision history

    ks	18. oct. 2008	rev 1.0
    	original version

    ks	20. oct. 2009	rev 1.1
    	unbenutzten code entfernt, all buffer base 0

    ks	20. dec. 2010	rev 1.2
    	parsing nach rfc1305

    ks	26. jul. 2011	rev 1.3
    	verbesserte ip-auswertung , neue fehlermeldung
    *)

    (*----------------------------------------------------------------------------------------------------------------*)
    (* Flags: 0x0100 (Standard query)                                                                                            *)
    (* 0... .... .... .... = Response: Message is a query                                                                   *)
    (* .000 0... ....  = Opcode: Standard query (0)                                                                          *)
    (* .... ..0. .... .... = Truncated: Message is not truncated                                                          *)
    (* .... ...1 .... .... = Recursion desired: Do query recursively                                                    *)
    (* .... .... .0.. .... = Z: reserved (0)                                                                                                  *)
    (* .... .... ...0 .... = Non-authenticated data OK: Non-authenticated data is unacceptable *)
    (*-----------------------------------------------------------------------------------------------------------------*)

    (*      0  1  2  3  4  5  6  7  8  9  0  1  2  3  4  5  *)
    (*    +--+--+--+--+--+--+--+--+--+--+--+--+--+--+--+--+ *)
    (*    |                      ID                       | idx: 0/1   *)
    (*    +--+--+--+--+--+--+--+--+--+--+--+--+--+--+--+--+ *)
    (*    |QR|   Opcode  |AA|TC|RD|RA|   Z    |   RCODE   | idx: 2/3   *)
    (*    +--+--+--+--+--+--+--+--+--+--+--+--+--+--+--+--+ *)
    (*    |                    QDCOUNT                    | idx: 4/5   *)
    (*    +--+--+--+--+--+--+--+--+--+--+--+--+--+--+--+--+ *)
    (*    |                    ANCOUNT                    | idx: 6/7   *)
    (*    +--+--+--+--+--+--+--+--+--+--+--+--+--+--+--+--+ *)
    (*    |                    NSCOUNT                    | idx: 8/9   *)
    (*    +--+--+--+--+--+--+--+--+--+--+--+--+--+--+--+--+ *)
    (*    |                    ARCOUNT                    | idx: 10/11 *)
    (*    +--+--+--+--+--+--+--+--+--+--+--+--+--+--+--+--+ *)

    (*
    Errorcodes  Description	References
    000	No ERROR. 		 	The request completed successfully.
    001	Format ERROR. 		The name server was unable to interpret the query.
    002	Server failure.  	The name server was unable to process this query due to a problem with the name server.
    003	Name ERROR. 	 	Meaningful only for responses from an authoritative name server, this code signifies that the DOMAIN name referenced in the query does not exist.
    004	Not Implemented. 	The name server does not support the requested kind of query.
    005	Refused. 			The name server refuses to perform the specified operation for policy reasons.
      						 For example, a name server may not wish to provide the information to the particular requester, or a name server may not wish to perform a particular operation (e.g., zone transfer) for particular data.
    006	YXDomain.			Name Exists when it should not.
    007	YXRRSet. RR			Set Exists when it should not.
    008	NXRRSet. RR			Set that should exist does not.
    009	NotAuth.			Server Not Authoritative for zone.
    010	NotZone,			Name not contained in zone.
    255	Timeout				No Response

    beispiel einer DNS Request von google.at
    ein request mit 3 Answer-Blocks

    DOMAIN Name System (response)
    [Request In: 3]
    [Time: 0.027533000 seconds]
    Transaction ID: 0x5e1a
    Flags: 0x8180 (Standard query response, No ERROR)
    1... .... .... .... = Response: Message is a response
    .000 0... .... .... = Opcode: Standard query (0)
    .... .0.. .... .... = Authoritative: Server is not an authority for DOMAIN
    .... ..0. .... .... = Truncated: Message is not truncated
    .... ...1 .... .... = Recursion desired: Do query recursively
    .... .... 1... .... = Recursion available: Server can do recursive queries
    .... .... .0.. .... = Z: reserved (0)
    .... .... ..0. .... = Answer authenticated: Answer/authority portion was not authenticated
    .... .... .... 0000 = Reply code: No ERROR (0)
    Questions: 1
    Answer RRs: 3
    Authority RRs: 0
    Additional RRs: 0

    Queries
    google.at: type A, class IN
    Name: google.at
    Type: A (Host address)
    Class: IN (0x0001)

    Answers
    google.at: type A, class IN, addr 72.14.221.104
    Name: google.at
    Type: A (Host address)
    Class: IN (0x0001)
    Time to live: 19 minutes, 9 seconds
    Data length: 4
    Addr: 72.14.221.104

    google.at: type A, class IN, addr 66.249.93.104
    Name: google.at
    Type: A (Host address)
    Class: IN (0x0001)
    Time to live: 19 minutes, 9 seconds
    Data length: 4
    Addr: 66.249.93.104

    google.at: type A, class IN, addr 216.239.59.104
    Name: google.at
    Type: A (Host address)
    Class: IN (0x0001)
    Time to live: 19 minutes, 9 seconds
    Data length: 4
    Addr: 216.239.59.104
    *)
END_FUNCTION_BLOCK

(* ---- DNS_DYN.st ---- *)
FUNCTION_BLOCK DNS_DYN
    (*http://www.oscat.de/images/OSCATNetwork/oscat_netlib121_en.pdf#page=92*)
    CASE state OF

    00:	IF ENABLE AND ((UPDATE AND NOT update_last) OR w.Q) THEN
    		state := 20;
    		DONE := FALSE;
    		BUSY := TRUE;
    		ERROR_C := DWORD#0;
    		ERROR_T := BYTE#0;

    		IF MODE = 0 THEN (* dyndns.org *)
    			s2 := CONCAT('http://members.dyndns.org/nic/UPDATE?HOSTNAME=',HOSTNAME);
    		ELSE (* selfhost.de *)
    			s2 := 'http://carol.selfhost.de/nic/UPDATE?HOSTNAME=1';
    		END_IF
    		IF IP4 > 0 THEN (* parametrierte IP verwenden *)
    			s1 := CONCAT('&myip=',IP4_TO_STRING(IP4));
    			s2 := CONCAT(s2,s1);
    		END_IF
    		URL_DATA:=STRING_TO_URL(STR:=s2, DEFAULT_PROTOCOL:='', DEFAULT_PATH:=''); (* URL for DNS UND HTTP-GET *)
    		s1 := CONCAT(USERNAME,':');
    		s1 := CONCAT(s1,PASSWORD); (* BASE64 Encode Text *)
    	END_IF

    20:	IF DNS_CLIENT.DONE THEN (* DNS_CLIENT *)
    			state := 40;
    	ELSIF (DNS_CLIENT.ERROR > DWORD#00) THEN (* Fehlerbehandlung *)
    		ERROR_C := DNS_CLIENT.ERROR;
    		ERROR_T := BYTE#01;
    		BUSY := FALSE;
    		state := 0;
    	END_IF

    40: IF base64_done THEN (* BASE64 Encode beendet ? *)
    		s1 := CONCAT('Authorization: Basic ',s2);
    		s1 := CONCAT(s1,'$0D$0AUser-Agent: x$0D$0A');
    		URL_DATA.HEADER := s1;
    		state := 60;
    	END_IF

    60:	IF HTTP_GET.DONE THEN
    		state := 0;
    		BUSY := FALSE;
    		DONE := TRUE;

    		(* !! Codes !!
    		Successful Updates: 		good , nchg
    		UPDATE Syntax Errors:		badsys , badagent
    		Account-Related Errors:		badauth , !donator
    		HOSTNAME-Related Errors:	notfqdn , nohost , !yours , numhost , abuse
    		Server Error Conditions:	dnserr , 911
    		*)
    		s2 := BUFFER_TO_STRING(PT:=ADR(R_BUF.BUFFER),SIZE:=SIZEOF(R_BUF.BUFFER),START:=HTTP_GET.BODY_START + 3,STOP:=HTTP_GET.BODY_STOP - 7);
    		IF FIND(s2,'good') = 0 THEN
    			IF FIND(s2,'nochg') = 0 THEN
    				ERROR_C := DWORD#1;
    				ERROR_T := BYTE#03;
    				DONE := FALSE;
    			END_IF
    		END_IF
    	ELSIF (HTTP_GET.ERROR > DWORD#00) THEN (* Fehlerbehandlung *)
    		ERROR_C := HTTP_GET.ERROR;
    		ERROR_T := BYTE#02;
    		BUSY := FALSE;
    		state := 0;
    	END_IF

    END_CASE

    DNS_CLIENT(IP_C:=IP_C,	S_BUF:=S_BUF, R_BUF:=R_BUF,DOMAIN:=URL_DATA.DOMAIN, IP4_DNS:=0, ACTIVATE:=state=20); (* DNS_CLIENT *)
    HTTP_GET( IP_C:=IP_C, S_BUF:=S_BUF, R_BUF:=R_BUF, IP4:=DNS_CLIENT.IP4, GET:=state=60, MODE:=2, UNLOCK_BUF:=state<>60,URL_DATA:=URL_DATA); (* HTTP_GET *)
    BASE64_ENCODE_STR( RUN:=state=40, STR1:=s1, STR2:=s2, DONE=>base64_done); (* BASE64 Encode *)

    IF T_UPDATE > T#0ms THEN w(IN:=state=0, PT:=T_UPDATE); END_IF
    update_last := UPDATE;

    (* revision history
    ks	01. jan. 2010	rev 1.0
    	original version

    *)
END_FUNCTION_BLOCK

(* ---- DNS_REV_CLIENT.st ---- *)
FUNCTION_BLOCK DNS_REV_CLIENT
    (*http://www.oscat.de/images/OSCATNetwork/oscat_netlib121_en.pdf#page=90*)
    (* DOMAIN Name System (query) *)

    CASE state OF
    00: (* auf positive Flanke GET warten *)
    	IF ACTIVATE AND NOT activate_last THEN
    		ERROR := DWORD#0;
    		ip4_copy := IP4; (* IP4 sichern *)
    		ip_state := BYTE#1;
    		DOMAIN := '';
    		DONE := FALSE;

    		d := '';
    		FOR i := 1 TO 4 DO
    			d := CONCAT(d,BYTE_TO_STRING(DWORD_TO_BYTE(IP4)));
    			d := CONCAT(d,'.');
    			IP4 := ROR(IP4,8);
    		END_FOR
    		d := CONCAT(d,'in-addr.arpa');
    		state := 10;
    	END_IF

    10: (* Bei IP_Control anmelden *)
    	IF ip_state = BYTE#3 THEN
    		dl := LEN(d);

    		(* sendebuffer initialisieren *)
    		char_count := 17 + dl;
    		FOR i := 0 TO char_count DO
    			S_BUF.BUFFER[i] := BYTE#00;
    		END_FOR

    		tid := UINT_TO_BYTE(BYTE_TO_UINT(tid) + UINT#1);
    		S_BUF.BUFFER[01] := tid; (* Transaction ID lowbyte *)
    		S_BUF.BUFFER[02] := BYTE#16#01; (* Flags: highbyte *)
    		S_BUF.BUFFER[05] := BYTE#16#01; (* Questions: lowbyte *)

    		(* den servernamen von hinten nach vorne bearbeiten *)
    		i := dl + 12;
    		char_count := 0;

    		WHILE i > 12 DO
    			char := CODE(STR:=d,POS:=i - 12);

    			(* prüfe auf haupt/sub domänen namens-teiler "." *)
    			IF char = BYTE#46 THEN
    				(* anstelle des teilers "." wird die länge des erkannten haupt/sub domänennames eingetragen *)
    				S_BUF.BUFFER[i] := INT_TO_BYTE(char_count);
    				char_count := 0;
    			ELSE
    				S_BUF.BUFFER[i] := char; (* char in buffer eintragen *)
    				char_count := char_count + 1; (* anzahl char zählen *)
    			END_IF
    			i := i - 1;
    		END_WHILE

    		S_BUF.BUFFER[i] := INT_TO_BYTE(char_count); (* längenangabe des ganz linken (ersten) domänennamens eintragen *)
    		i := dl + 15; (* position hinter dem servernamen *)
    		S_BUF.BUFFER[i] := BYTE#12; (* Type: PTR (DOMAIN name pointer) lowbyte *)
    		i := i + 2;
    		S_BUF.BUFFER[i] := BYTE#01; (* Class: IN lowbyte *)
    		i := i + 1;

    		(* IP Datenverkehr einrichten *)
    		IP_C.C_PORT := WORD#53; (* Portnummer eintragen *)
    		IP_C.C_IP := IP4_DNS; (* IP eintragen *)
    		IP_C.C_MODE := BYTE#1; (* Mode: UDP+AKTIV+PORT+IP *)
    		IP_C.C_ENABLE := TRUE; (* Verbindungsaufbau freigeben *)
    		IP_C.TIME_RESET := TRUE; (* Zeitueberwachung rücksetzen *)
    		IP_C.R_OBSERVE  := TRUE; (* Datenempfang ueberwachen *)
    		S_BUF.SIZE := INT_TO_UINT(i); (* sendelänge eintragen *)
    		R_BUF.SIZE := UINT#0; (* Empfangslänge rücksetzen *)
    		state := 30;
    	END_IF

    30:
    	IF IP_C.ERROR <> DWORD#00 THEN
    		ERROR := IP_C.ERROR;
    	(* prüfe ob antwort telegramm die richtige Transaction-ID und mindestlänge hat *)
    	ELSIF (S_BUF.SIZE = UINT#0) AND (tid = R_BUF.BUFFER[1]) AND (R_BUF.SIZE >= INT_TO_UINT(i+12)) THEN

    		(* prüfe Return code der Flags. 4 bits *)
    		ERROR := BYTE_TO_DWORD(R_BUF.BUFFER[3] AND BYTE#2#0000_1111);

    		IF ERROR = DWORD#00 THEN

    			i := R_BUF.SIZE - 2;
    			WHILE R_BUF.BUFFER[i] > 0 DO
    				IF i = 0 THEN EXIT; END_IF
    				i := i - 1;
    			END_WHILE

    			i := i + 2;
    			p1 := i + 1;
    			WHILE i < R_BUF.SIZE DO
    				dl := R_BUF.BUFFER[i];
    				IF dl > 0 THEN
    					R_BUF.BUFFER[i] := BYTE#46;
    					i := i + dl + 1;
    				ELSE
    					DOMAIN := BUFFER_TO_STRING(PT:=ADR(R_BUF.BUFFER),SIZE:=SIZEOF(R_BUF.BUFFER),START:=p1,STOP:=i-1);
    					EXIT;
    				END_IF
    			END_WHILE
    			state := 0;
    			DONE := TRUE;
    		END_IF
    	END_IF

    	IF ERROR <> DWORD#0 THEN
    		state := 0;
    	END_IF

    	IF state = 0 THEN
    		IP_C.R_OBSERVE := FALSE; (* Datenempfang ueberwachen *)
    		ip_state := BYTE#4; (* Abmelden *)
    	END_IF

    END_CASE

    activate_last := ACTIVATE; (* letzten Status sichern zur Flankenerkennung *)

    (* IP_FIFO *)
    IP_FIFO(FIFO:=IP_C.FIFO,state:=ip_state,ID:=ip_id);

    (* revision history

    ks	28. dec. 2009	rev 1.0
    	original version

    *)

    (*----------------------------------------------------------------------------------------------------------------*)
    (* Flags: 0x0100 (Standard query)                                                                                            *)
    (* 0... .... .... .... = Response: Message is a query                                                                   *)
    (* .000 0... ....  = Opcode: Standard query (0)                                                                          *)
    (* .... ..0. .... .... = Truncated: Message is not truncated                                                          *)
    (* .... ...1 .... .... = Recursion desired: Do query recursively                                                    *)
    (* .... .... .0.. .... = Z: reserved (0)                                                                                                  *)
    (* .... .... ...0 .... = Non-authenticated data OK: Non-authenticated data is unacceptable *)
    (*-----------------------------------------------------------------------------------------------------------------*)

    (*
    Errorcodes  Description	References
    000	No ERROR. 		 	The request completed successfully.
    001	Format ERROR. 		The name server was unable to interpret the query.
    002	Server failure.  	The name server was unable to process this query due to a problem with the name server.
    003	Name ERROR. 	 	Meaningful only for responses from an authoritative name server, this code signifies that the DOMAIN name referenced in the query does not exist.
    004	Not Implemented. 	The name server does not support the requested kind of query.
    005	Refused. 			The name server refuses to perform the specified operation for policy reasons.
      						 For example, a name server may not wish to provide the information to the particular requester, or a name server may not wish to perform a particular operation (e.g., zone transfer) for particular data.
    006	YXDomain.			Name Exists when it should not.
    007	YXRRSet. RR			Set Exists when it should not.
    008	NXRRSet. RR			Set that should exist does not.
    009	NotAuth.			Server Not Authoritative for zone.
    010	NotZone,			Name not contained in zone.
    255	Timeout				No Response
    *)
END_FUNCTION_BLOCK

(* ---- FILE_BLOCK.st ---- *)
FUNCTION_BLOCK FILE_BLOCK
    (*http://www.oscat.de/images/OSCATNetwork/oscat_netlib121_en.pdf#page=152*)
    CASE step OF
    0:	IF MODE > 0 THEN
    		ERROR := 0;
    		IF FSD.FILE_OPEN AND (FSD.FILE_SIZE = 0 OR POS >= FSD.FILE_SIZE) THEN
    			ERROR := 255;
    			MODE := 0;
    		ELSIF POS < data_start OR POS > data_stop OR NOT FSD.FILE_OPEN THEN (* Daten lesen notwendig *)
    			FSD.FILENAME := FILENAME;
    			FSD.MODE := 1; (* open + read *)
    			FSD.OFFSET := POS;
    			PT.SIZE := 65535; (* maximale anzahl lesen *);
    			data_start := 0;
    			data_stop := 0;
    			step := 10;
    		ELSE (* Daten sind im Buffer vorhanden *)
    			i := UDINT_TO_INT(POS - data_start); (* index berechnen *)
    			DATA := PT.BUFFER[i];
    			MODE := 0;
    			(* ---------------------- Debug-Message ----------------------------*)
    			(*IF _debug_enable THEN
    				LOG_CL.NEW_MSG := 'FB: POS: ~1 Byte: ~2 >~3<';
    				LOG_CL.PRINTF[1] := UDINT_TO_STRING(POS);
    				LOG_CL.PRINTF[2] := BYTE_TO_STRING(DATA);
    				LOG_CL.PRINTF[3] := CHR_TO_STRING(DATA);
    				LOG_MSG();
    			END_IF*)
    			(* -----------------------------------------------------------------*)
    		END_IF
    	END_IF

    10:	IF FSD.MODE = 0 THEN (* Befehl beendet *)
    		IF FSD.ERROR > 0 THEN
    			ERROR := FSD.ERROR; (* Fehler ausgeben *)
    			MODE := 0;
    		ELSE
    			data_start := POS;
    			data_stop := POS + UINT_TO_UDINT(PT.SIZE) - 1;
    		END_IF
    		step := 0;
    	END_IF
    END_CASE

    (* revision history
    ks	23. sep. 2010	rev 1.0
    	original version
    *)
END_FUNCTION_BLOCK

(* ---- FILE_SERVER.st ---- *)
FUNCTION_BLOCK FILE_SERVER
    (*http://www.oscat.de/images/OSCATNetwork/oscat_netlib121_en.pdf#page=154*)
    CASE step OF
    0:
    	IF FSD.MODE = LIMIT(1,FSD.MODE,5) THEN

    		(* ---------------------- Debug-Message ----------------------------*)
    		(*IF _debug_enable THEN
    			LOG_CL.NEW_MSG := 'File_Start Mode=~1';
    			LOG_CL.PRINTF[1] := BYTE_TO_STRING(FSD.MODE);
    			FB_LOG_MESSAGE();
    		END_IF*)
    		(* -----------------------------------------------------------------*)

    		buf_size := SIZEOF(PT.BUFFER);

    		IF FSD.MODE = 4 THEN (* File_Remove *)
    			IF handle > 0 THEN
    				file_change := TRUE;
    				step := 32000; (* File_Close ausführen *)
    			ELSE
    				step := 90; (* File_Remove ausführen *)
    			END_IF

    		ELSIF FSD.MODE = 5 THEN (* File_Close *)
    			step := 32000; (* File_Close ausführen *)

    		ELSIF handle = 0 THEN (* MODE 1,2,3 *)
    			step := 100; (* File muss erst geöffnet werden *)

    		ELSE (* File ist geöffnset *)
    			IF used_filename = FSD.FILENAME AND FSD.MODE = last_mode THEN (* kein Moduswechsel ? *)
    				step := 200; (* ohne open prozedure weitermachen *)
    			ELSE
    				step := 32000;
    				file_change := TRUE;
    			END_IF
    		END_IF
    	END_IF

    (* ----------------------------------- *)
    090: (* File_Remove *)
    	command := 7; (* File Remove *)
    	step := 95;

    095: (* File_Remove beendet *)
    	IF command = 0 THEN
    		step := 30000; (* Beenden *)
    	END_IF
    (* ----------------------------------- *)

    100: (* File Size - Dateigroesse bestimmen *)
    	command := 8; (* File Size *)
    	step := 110;

    110: (* File Size beendet *)
    	IF command = 0 THEN
    		IF FSD.MODE = 1 THEN (* open + read *)
    			open_mode := 'r';
    			FSD.file_size := file_size; (* aktuelle Dateigroesse *)
    		ELSIF FSD.MODE = 2 THEN (* open + write *)
    			open_mode := 'a';
    			FSD.file_size := file_size; (* aktuelle Dateigroesse *)
    		ELSE (* open new + write *)
    			open_mode := 'w';
    			FSD.file_size := 0; (* aktuelle Dateigroesse *)
    		END_IF
    		command := 1; (* File Open *)
    		last_mode := FSD.MODE;
    		step := 150; (* File_Open ausführen *)
    	END_IF

    150: (* File Open *)
    	IF command = BYTE#0 THEN
    		IF error THEN
    			step := 30000; (* Beenden *)
    		ELSE
    			(* Filedaten eintragen *)
    			handle := open_handle;
    			used_filename := FSD.FILENAME;
    			file_position := UDINT#4294967295; (* maximal = unbekannt *)
    			FSD.FILE_OPEN := TRUE;
    			step := 200;
    		END_IF
    	END_IF

    200: (* File Seek *)
    	IF FSD.OFFSET = UDINT#4294967294 THEN (* 16#FFFF_FFFE -> Zeiger auf Dateiende stellen *)
    		command := 5; (* File-Seek *)
    		seek_position := FSD.file_size;
    		step := 210;
    	ELSIF FSD.OFFSET > FSD.file_size THEN (* prüfe auf gültige offset-vorgabe *)
    		error_code := 255;
    		step := 30000; (* Beenden *)
    	ELSIF FSD.OFFSET <> file_position THEN
    		command := 5; (* File-Seek *)
    		seek_position := FSD.OFFSET;
    		step := 210;
    	ELSE
    		step := 300;
    	END_IF

    210: (* File Seek *)
    	IF command = 0 THEN
    		file_position := seek_position;
    		IF error THEN
    			step := 30000; (* Beenden *)
    		ELSE
    			step := 300;
    		END_IF
    	END_IF

    300: (* Read or Write ? *)
    	IF FSD.MODE = 1 THEN
    		step := 400; (* Read *)
    	ELSE
    		step := 500; (* Write *)
    	END_IF

    400: (* File Read *)
    	IF UINT_TO_UDINT(PT.SIZE) > buf_size THEN (* Leselänge auf Buffergroesse begrenzen *)
    		read_max_length := buf_size;
    	ELSE
    		read_max_length := UINT_TO_UDINT(PT.SIZE);
    	END_IF

    	(* Leselänge an Dateilänge anpassen *)
    	IF file_position + read_max_length > FSD.file_size THEN
    		read_max_length := FSD.file_size - file_position;
    	END_IF

    	IF read_max_length > 0 THEN
    		command := 3; (* File_Read *)
    		step := 410;
    	ELSE
    		PT.SIZE := UINT#0;
    		step := 30000; (* Beenden *)
    	END_IF

    410: (* File Read *)
    	IF command = 0 THEN
    		PT.SIZE := UDINT_TO_UINT(length_read);
    		IF NOT error THEN
    			file_position := file_position + length_read; (* aktueller file_position korrigieren *)
    			FSD.OFFSET := file_position;
    		END_IF
    		step := 30000; (* Beenden *)
    	END_IF

    500: (* File Write *)
    	IF UINT_TO_UDINT(PT.SIZE) > buf_size THEN (* Schreiblänge auf Buffergroesse begrenzen *)
    		write_length := buf_size;
    	ELSE
    		write_length := UINT_TO_UDINT(PT.SIZE);
    	END_IF

    	IF write_length > 0 THEN
    		command := 4; (* File_Write *)
    		step := 510;
    	ELSE
    		step := 30000; (* Beenden *)
    	END_IF

    510:
    	IF command = 0 THEN
    		IF NOT error THEN
    			file_position := file_position + length_written; (* aktueller file_position korrigieren *)
    			FSD.OFFSET := file_position;
    			IF file_position > FSD.file_size THEN (* Datei ist groesser geworden *)
    				FSD.file_size := file_position;
    			END_IF
    		END_IF
    		step := 30000; (* Beenden *)
    	END_IF

     (* --------------------------------------------- *)

    30000: (* Befehl fertig *)
    	FSD.MODE := 0;
    	FSD.error := error_code;
    	step := 0;

    	(* ---------------- Debug-Message -----------------------*)
    	(*IF _debug_enable THEN
    		LOG_CL.NEW_MSG := 'File_Stop: File ~1, error ~7, code ~8';
    		LOG_CL.PRINTF[1]  := used_filename;
    		LOG_CL.PRINTF[7]  := INT_TO_STRING(BOOL_TO_INT(error));
    		LOG_CL.PRINTF[8]  := BYTE_TO_STRING(error_code);
    		FB_LOG_MESSAGE();
    	END_IF*)
    	(* --------------------------------------------- *)

    32000:
    	IF handle > 0 THEN
    		command := 2; (* File_Close ausführen *)
    	END_IF
    	step := 32100;

    32100:
    	IF command = 0 THEN (* File Close beendet *)
    		(* Filedaten ablöschen *)
    		FSD.FILE_OPEN := FALSE;
    		file_position := 0;
    		FSD.file_size := 0;
    		FSD.OFFSET := 0;
    		used_filename := '';
    		handle := 0;

    		(* File_Name wurde fliegend geändert ? *)
    		IF file_change THEN
    			file_change := FALSE;
    			step := 0;
    		ELSE
    			step := 30000;
    		END_IF
    	END_IF

    END_CASE

    (* 1 = file_open
       2 = file_close
       3 = file_read
       4 = file_write
       5 = file_seek
       6 = file_tell
       7 = file_remove
    *)

    FSR(MODE:=BYTE#0,command:=command,FSD:=FSD); (* File server Runtime / Befehlsstart überwachen *)

    (* ------------ File Open ------------- *)
    IF command = 1 THEN
    	open_handle := SysFileOpen(FSD.FILENAME,open_mode);
    	error := open_handle = 0;
    	error_code := SEL(error,0,command);
    	command := 0;
    	FSR(MODE:=BYTE#1,command:=command,FSD:=FSD); (* File server Runtime / Befehlstop überwachen *)
    	(* ---------------- Debug-Message -----------------------*)
    	(*IF _debug_enable THEN
    		LOG_CL.NEW_MSG := 'Open: File ~1, handle ~2 , mode ~3 , error ~7, code ~8';
    		LOG_CL.PRINTF[1] := FSD.FILENAME;
    		LOG_CL.PRINTF[2] := DWORD_TO_STRING(open_handle);
    		LOG_CL.PRINTF[3] := open_mode;
    		LOG_CL.PRINTF[7] := INT_TO_STRING(BOOL_TO_INT(error));
    		LOG_CL.PRINTF[8] := BYTE_TO_STRING(error_code);
    		FB_LOG_MESSAGE();
    	END_IF*)
    	(* -----------------------------------------------------------------*)
    END_IF

    (* ----------- File Close ------------- *)
    IF command = 2 THEN
    	error := NOT SysFileClose(handle);
    	error_code := SEL(error,0,command);
    	command := 0;
    	FSR(MODE:=BYTE#1,command:=command,FSD:=FSD); (* File server Runtime / Befehlstop überwachen *)
    	(* ---------------- Debug-Message -----------------------*)
    	(*IF _debug_enable THEN
    		LOG_CL.NEW_MSG := 'Close: File ~1, error ~7, code ~8';
    		LOG_CL.PRINTF[1] := used_filename;
    		LOG_CL.PRINTF[7] := INT_TO_STRING(BOOL_TO_INT(error));
    		LOG_CL.PRINTF[8] := BYTE_TO_STRING(error_code);
    		FB_LOG_MESSAGE();
    	END_IF*)
    	(* -----------------------------------------------------------------*)
    END_IF

    (* ------------ File Read ------------- *)
    IF command = 3 THEN
    	length_read := SysFileRead(handle, ADR(PT.BUFFER), read_max_length);
    	error := length_read = 0;
    	error_code := SEL(error,0,command);
    	command := 0;
    	FSR(MODE:=BYTE#1,command:=command,FSD:=FSD); (* File server Runtime / Befehlstop überwachen *)
    	(* ---------------- Debug-Message -----------------------*)
    	(*IF _debug_enable THEN
    		LOG_CL.NEW_MSG := 'Read: File ~1, soll ~2,ist ~3 ,error ~7, code ~8';
    		LOG_CL.PRINTF[1] := used_filename;
    		LOG_CL.PRINTF[2] := UDINT_TO_STRING(read_max_length);
    		LOG_CL.PRINTF[3] := UDINT_TO_STRING(length_read);
    		LOG_CL.PRINTF[7] := INT_TO_STRING(BOOL_TO_INT(error));
    		LOG_CL.PRINTF[8] := BYTE_TO_STRING(error_code);
    		FB_LOG_MESSAGE();
    	END_IF*)
    	(* -----------------------------------------------------------------*)
    END_IF

    (* ------------ File Write ------------- *)
    IF command = 4 THEN
    	length_written := SysFileWrite(handle, ADR(PT.BUFFER), write_length);
    	error := length_written = 0;
    	error_code := SEL(error,0,command);
    	command := 0;
    	FSR(MODE:=BYTE#1,command:=command,FSD:=FSD); (* File server Runtime / Befehlstop überwachen *)
    	(* ---------------- Debug-Message -----------------------*)
    	(*IF _debug_enable THEN
    		LOG_CL.NEW_MSG := 'Write: File ~1, soll ~2,ist ~3 ,error ~7, code ~8';
    		LOG_CL.PRINTF[1] := used_filename;
    		LOG_CL.PRINTF[2] := UDINT_TO_STRING(write_length);
    		LOG_CL.PRINTF[3] := UDINT_TO_STRING(length_written);
    		LOG_CL.PRINTF[7] := INT_TO_STRING(BOOL_TO_INT(error));
    		LOG_CL.PRINTF[8] := BYTE_TO_STRING(error_code);
    		FB_LOG_MESSAGE();
    	END_IF*)
    	(* -----------------------------------------------------------------*)
    END_IF

    (* ------------ File Seek ------------- *)
    IF command = 5 THEN
    	error := NOT SysFileSetPos(handle, seek_position);
    	error_code := SEL(error,0,command);
    	command := 0;
    	FSR(MODE:=BYTE#1,command:=command,FSD:=FSD); (* File server Runtime / Befehlstop überwachen *)
    	(* ---------------- Debug-Message -----------------------*)
    	(*IF _debug_enable THEN
    		LOG_CL.NEW_MSG := 'Seek: File ~1,pos ~3 ,error ~7, code ~8';
    		LOG_CL.PRINTF[1] := used_filename;
    		LOG_CL.PRINTF[3] := UDINT_TO_STRING(seek_position);
    		LOG_CL.PRINTF[7] := INT_TO_STRING(BOOL_TO_INT(error));
    		LOG_CL.PRINTF[8] := BYTE_TO_STRING(error_code);
    		FB_LOG_MESSAGE();
    	END_IF*)
    	(* -----------------------------------------------------------------*)
    END_IF

    (* ------------ File Tell ------------- *)
    IF command = 6 THEN
    	tell_position := SysFileGetPos(handle);
    	error := tell_position < 0;
    	error_code := SEL(error,0,command);
    	command := 0;
    	FSR(MODE:=BYTE#1,command:=command,FSD:=FSD); (* File server Runtime / Befehlstop überwachen *)
    	(* ---------------- Debug-Message -----------------------*)
    	(*IF _debug_enable THEN
    		LOG_CL.NEW_MSG := 'Tell: File ~1, pos ~3 ,error ~7, code ~8';
    		LOG_CL.PRINTF[1] := used_filename;
    		LOG_CL.PRINTF[3] := UDINT_TO_STRING(tell_position);
    		LOG_CL.PRINTF[7] := INT_TO_STRING(BOOL_TO_INT(error));
    		LOG_CL.PRINTF[8] := BYTE_TO_STRING(error_code);
    		FB_LOG_MESSAGE();
    	END_IF*)
    	(* -----------------------------------------------------------------*)
    END_IF

    (* ------------ File Remove ------------- *)
    IF command = 7 THEN
    	error := NOT SysFileDelete(FSD.FILENAME);
    	error_code := SEL(error,0,command);
    	command := 0;
    	FSR(MODE:=BYTE#1,command:=command,FSD:=FSD); (* File server Runtime / Befehlstop überwachen *)
    	(* ---------------- Debug-Message -----------------------*)
    	(*IF _debug_enable THEN
    		LOG_CL.NEW_MSG := 'Remove: File ~1, error ~7, code ~8';
    		LOG_CL.PRINTF[1] := FSD.FILENAME;
    		LOG_CL.PRINTF[7] := INT_TO_STRING(BOOL_TO_INT(error));
    		LOG_CL.PRINTF[8] := BYTE_TO_STRING(error_code);
    		FB_LOG_MESSAGE();
    	END_IF*)
    	(* -----------------------------------------------------------------*)
    END_IF

    (* ------------ File Size ------------- *)
    IF command = 8 THEN
    	file_size := SysFileGetSize(FSD.FILENAME);
    	error_code := 0; (* kein Errorcode vorhanden *)
    	command := 0;
    	FSR(MODE:=BYTE#1,command:=command,FSD:=FSD); (* File server Runtime / Befehlstop überwachen *)
    	(* ---------------- Debug-Message -----------------------*)
    	(*IF _debug_enable THEN
    		LOG_CL.NEW_MSG := 'Size: File ~1, size ~3, error ~7, code ~8';
    		LOG_CL.PRINTF[1] := FSD.FILENAME;
    		LOG_CL.PRINTF[3] := DINT_TO_STRING(file_size);
    		LOG_CL.PRINTF[7] := INT_TO_STRING(BOOL_TO_INT(error));
    		LOG_CL.PRINTF[8] := BYTE_TO_STRING(error_code);
    		FB_LOG_MESSAGE();
    	END_IF*)
    	(* -----------------------------------------------------------------*)
    END_IF

    (* ---------------- Debug-Message -----------------------*)
    (*IF _debug_enable THEN
    	IF step_last <> step THEN
    		LOG_CL.NEW_MSG := 'step: ~1';
    		LOG_CL.PRINTF[1] := INT_TO_STRING(step);
    		FB_LOG_MESSAGE();
    	END_IF
    	step_last := step;
    END_IF*)
    (* -----------------------------------------------------------------*)

    (* revision history
    ks	08. mar. 2016	rev 1.2
    	Filesystem Laufzeitmessungen

    ks	02. oct. 2014	rev 1.1.1
    	PCWORX SRT File Delete error

    ks	05. mai. 2012	rev 1.1
    	auto_close funktion entfernt

    ks	23. sep. 2010	rev 1.0
    	original version
    *)
END_FUNCTION_BLOCK

(* ---- FILE_SERVER_RUNTIME.st ---- *)
FUNCTION_BLOCK FILE_SERVER_RUNTIME
    (*http://www.oscat.de/images/OSCATBasic/oscat_basic333_en.pdf#page=154*)
    IF init = FALSE THEN
    	init := TRUE;
    	FSD.runtime.TIME_FILE_OPEN_MIN := UDINT#99999999;
    	FSD.runtime.TIME_FILE_CLOSE_MIN := UDINT#99999999;
    	FSD.runtime.TIME_FILE_READ_MIN := UDINT#99999999;
    	FSD.runtime.TIME_FILE_WRITE_MIN := UDINT#99999999;
    	FSD.runtime.TIME_FILE_TELL_MIN := UDINT#99999999;
    	FSD.runtime.TIME_FILE_SEEK_MIN := UDINT#99999999;
    	FSD.runtime.TIME_FILE_DELETE_MIN := UDINT#99999999;
    END_IF

    (* warten auf File_Server Befehl *)
    IF MODE = BYTE#0 THEN

    	(* neuen befehl erkannt *)
    	IF last_command = BYTE#0 AND COMMAND <> BYTE#0 THEN

    		(* read system time *)
    		start_tx := T_PLC_MS();

    	END_IF
    END_IF

    IF MODE = BYTE#1 THEN

    	(* read system time *)
    	stop_tx:=  T_PLC_MS();

    	runtime:= (stop_tx - start_tx);

    	CASE BYTE_TO_INT(COMMAND) OF

    	1:	FSD.runtime.TIME_FILE_OPEN_CUR := runtime; 			(* aktuelle laufzeit *)
    		IF FSD.runtime.TIME_FILE_OPEN_MAX < runtime THEN
    			FSD.runtime.TIME_FILE_OPEN_MAX := runtime;		(* neue max laufzeit *)
    		END_IF
    		IF FSD.runtime.TIME_FILE_OPEN_MIN > runtime THEN
    			FSD.runtime.TIME_FILE_OPEN_MIN := runtime;		(* neue min laufzeit *)
    		END_IF

    	2:	FSD.runtime.TIME_FILE_CLOSE_CUR := runtime; 			(* aktuelle laufzeit *)
    		IF FSD.runtime.TIME_FILE_CLOSE_MAX < runtime THEN
    			FSD.runtime.TIME_FILE_CLOSE_MAX := runtime;		(* neue max laufzeit *)
    		END_IF
    		IF FSD.runtime.TIME_FILE_CLOSE_MIN > runtime THEN
    			FSD.runtime.TIME_FILE_CLOSE_MIN := runtime;		(* neue min laufzeit *)
    		END_IF

    	3:	FSD.runtime.TIME_FILE_READ_CUR := runtime; 			(* aktuelle laufzeit *)
    		IF FSD.runtime.TIME_FILE_READ_MAX < runtime THEN
    			FSD.runtime.TIME_FILE_READ_MAX := runtime;		(* neue max laufzeit *)
    		END_IF
    		IF FSD.runtime.TIME_FILE_READ_MIN > runtime THEN
    			FSD.runtime.TIME_FILE_READ_MIN := runtime;		(* neue min laufzeit *)
    		END_IF

    	4:	FSD.runtime.TIME_FILE_WRITE_CUR := runtime; 			(* aktuelle laufzeit *)
    		IF FSD.runtime.TIME_FILE_WRITE_MAX < runtime THEN
    			FSD.runtime.TIME_FILE_WRITE_MAX := runtime;		(* neue max laufzeit *)
    		END_IF
    		IF FSD.runtime.TIME_FILE_WRITE_MIN > runtime THEN
    			FSD.runtime.TIME_FILE_WRITE_MIN := runtime;		(* neue min laufzeit *)
    		END_IF

    	5:	FSD.runtime.TIME_FILE_SEEK_CUR := runtime; 			(* aktuelle laufzeit *)
    		IF FSD.runtime.TIME_FILE_SEEK_MAX < runtime THEN
    			FSD.runtime.TIME_FILE_SEEK_MAX := runtime;		(* neue max laufzeit *)
    		END_IF
    		IF FSD.runtime.TIME_FILE_SEEK_MIN > runtime THEN
    			FSD.runtime.TIME_FILE_SEEK_MIN := runtime;		(* neue min laufzeit *)
    		END_IF

    	6:	FSD.runtime.TIME_FILE_TELL_CUR := runtime; 			(* aktuelle laufzeit *)
    		IF FSD.runtime.TIME_FILE_TELL_MAX < runtime THEN
    			FSD.runtime.TIME_FILE_TELL_MAX := runtime;		(* neue max laufzeit *)
    		END_IF
    		IF FSD.runtime.TIME_FILE_TELL_MIN > runtime THEN
    			FSD.runtime.TIME_FILE_TELL_MIN := runtime;		(* neue min laufzeit *)
    		END_IF

    	7:	FSD.runtime.TIME_FILE_DELETE_CUR := runtime; 			(* aktuelle laufzeit *)
    		IF FSD.runtime.TIME_FILE_DELETE_MAX < runtime THEN
    			FSD.runtime.TIME_FILE_DELETE_MAX := runtime;		(* neue max laufzeit *)
    		END_IF
    		IF FSD.runtime.TIME_FILE_DELETE_MIN > runtime THEN
    			FSD.runtime.TIME_FILE_DELETE_MIN := runtime;		(* neue min laufzeit *)
    		END_IF

    	END_CASE

    END_IF

    last_command := COMMAND;

    (* revision history

    ks	08. mar. 2016	rev 1.0
    	original version
    *)
END_FUNCTION_BLOCK

(* ---- FTP_CLIENT.st ---- *)
FUNCTION_BLOCK FTP_CLIENT
    (*http://www.oscat.de/images/OSCATNetwork/oscat_netlib121_en.pdf#page=94*)
    CASE step OF

    00:	IF ACTIVATE AND NOT activate_last THEN
    		ftp_file_size := UDINT#0;
    		TIMEOUT := MAX(T#10s,TIMEOUT);
    		timeout2 := TIMEOUT + T#1s;
    		timeout3 := TIMEOUT / 2;
    		DONE := FALSE;
    		ip_c1_red_disable := FALSE;
    		ip_c2_red_disable := FALSE;
    		ERROR_C := DWORD#0;
    		ERROR_T := BYTE#0;
    		FSD.ERROR := BYTE#0;
    		URL_DATA := STRING_TO_URL(STR:=FTP_URL,DEFAULT_PROTOCOL:='',DEFAULT_PATH:='/');
    		IF LEN(URL_DATA.USER) = 0 THEN
    			URL_DATA.USER := 'Anonymous';
    			URL_DATA.PASSWORD := 'User@';
    		END_IF

    		FILE_PATH_SPLIT(FILENAME:=FILENAME,X:=fpd); (* Datei-Path zerlegen *)
    		str1 := fpd.FILENAME; (* zwischenspeichern *)
    		FILE_PATH_SPLIT(FILENAME:=URL_DATA.PATH,X:=fpd); (* FTP-Path zerlegen *)
    		IF LEN(fpd.FILENAME) = 0 THEN (* wenn FTP-Path keinen Dateinamen enthält , dann den Namen der lokalen Datei benutzen *)
    			ftp_path := CONCAT(URL_DATA.PATH,str1);
    		ELSE
    			ftp_path := URL_DATA.PATH;
    		END_IF
    		step := 10;
    	END_IF

    10:	IF DNS_CLIENT.DONE THEN
    		step := 20;
    	ELSIF DNS_CLIENT.ERROR <> DWORD#0 THEN
    		ERROR_C := DNS_CLIENT.ERROR;
    		ERROR_T := BYTE#1;
    		step := 980;
    	END_IF

    20:	(* FTP Steuerkanal einrichten *)
    	IP_C1.C_PORT := WORD#21; (* Portnummer eintragen *)
      	IP_C1.C_IP := DNS_CLIENT.IP4; (* IP eintragen *)
      	IP_C1.C_MODE := BYTE#0; (* Mode: TCP+ACTIV+PORT *)
      	IP_C1.TIME_RESET := TRUE; (* Zeitueberwachung rücksetzen *)
      	IP_C1.C_ENABLE := TRUE; (* Verbindungsaufbau freigeben *)
      	IP_C1.R_OBSERVE := TRUE; (* Empfangsueberwachung *)
    	R_BUF1.SIZE := UINT#0;

      	IP_C2.C_ENABLE   := FALSE; (* Verbindungsaufbau sperren *)
    	step := 30;

    30:	IF rcv_state = 220 THEN (* 220 = Service ready for new user *)
    		snd_text := CONCAT('USER ',URL_DATA.USER);
    		next_step := 40;
    	END_IF

    40:	IF rcv_state = 331 THEN (* 331 = User name okay, need password *)
    		snd_text := CONCAT('PASS ',URL_DATA.PASSWORD);
    		next_step := 50;
    	ELSIF rcv_state = 230 THEN (* 230 = User logged in, proceed *)
    		next_step := 50;
    	ELSIF rcv_state = 220 THEN (* 220 = Service ready for new user *)
    		next_step := 20; (* WORK verbindung sollte ab/aufgebaut werden *)
    	END_IF

    50:	IF rcv_state = 230 THEN (* 230 = User logged in, proceed *)
    		snd_text := 'TYPE I';  (* binären Modus aktivieren *)
    		next_step := 54;
    	END_IF

    54:	IF rcv_state = 200 THEN (* 200 = Command okay *)
    		IF FTP_DOWNLOAD THEN (* Datei von FTP Empfangen *)
    			snd_text := CONCAT('SIZE ', ftp_path); (* SIZE /PFAD/FILENAME *)
    			next_step := 56;
    		ELSE
    			step := 60;
    		END_IF
    	END_IF

    56:	IF rcv_state = 213 THEN (* 213 Filesize *)
    		str1 := ELEMENT_GET(SEP:=BYTE#32,POS:=1,ELEMENT:=rcv_text);
    		ftp_file_size := STRING_TO_UDINT(str1); (* Dateigroesse in bytes gestimmen *)
    		step := 60;
    	END_IF

    60:	IF FTP_ACTIV THEN (* FTP Server aktiv *)
    		IF URL_DATA.PORT = WORD#0 THEN
    			URL_DATA.PORT := WORD#20; (* Standard Datenkanal *)
    		END_IF
    		str2 := '';
    		dw_tmp := PLC_IP4;
    		FOR idx1 := 0 TO 5 DO
    			IF idx1 = 4 THEN
    				dw_tmp := ROR(WORD_TO_DWORD(URL_DATA.PORT),8);
    			ELSE
    				dw_tmp := ROL(dw_tmp,8);
    			END_IF
    			str2 := CONCAT(str2,BYTE_TO_STRING(DWORD_TO_BYTE(dw_tmp)));
    			IF idx1 < 5 THEN
    				str2 := CONCAT(str2,',');
    			END_IF
    		END_FOR
    		dw_tmp := DNS_CLIENT.IP4; (* IP eintragen *)
    		w_tmp := URL_DATA.PORT; (* Port Nummer des Datenkanals *)
    		snd_text := CONCAT('PORT ',str2); (* FTP Server in den aktiv-mode schalten *)
    		next_step := 80;
    	ELSE
    		snd_text := 'PASV';  (* FTP Server in den passiv-mode schalten *)
    		next_step := 70;
    	END_IF
    	step := 999; (* Warten auf next_step *)

    70:	IF rcv_state = 227 THEN (* 227 = Entered Passive Mode (213,202,225,43,212,186) *)
    		idx1 := FIND(rcv_text , '(' );
    		idx2 := FIND(rcv_text , ')' );
    		IF idx1 > 0 AND idx2 > idx1+1 THEN
    			str1 := MID(rcv_text, idx2 - idx1 - 1, idx1+1);
    			FOR idx1 := 0 TO 5 DO
    				str2 := ELEMENT_GET(SEP:=BYTE#44,POS:=idx1,ELEMENT:=str1);
    				byar[idx1] := STRING_TO_BYTE(str2);
    			END_FOR
    			dw_tmp := DWORD_OF_BYTE(byar[0],byar[1],byar[2],byar[3]); (* IP Adresse des Datenkanals *)
    			w_tmp := WORD_OF_BYTE(byar[4],byar[5]); (* Port Nummer des Datenkanals *)
    		END_IF
    		step := 100;
    	END_IF

    80:	IF rcv_state = 200 THEN (* 200 = PORT command successful *)
    		step := 100;
    	END_IF

    100:IP_C2.C_MODE := SEL(FTP_ACTIV,BYTE#0,BYTE#2); (* Aktiv = Mode 2: TCP+PASSIV+PORT / passiv = Mode 0: TCP+ACTIV+PORT *)
    	IP_C2.C_IP := dw_tmp; (* IP Adresse des Datenkanals *)
    	IP_C2.C_PORT := w_tmp; (* Port Nummer des Datenkanals *)
      	IP_C2.TIME_RESET := TRUE; (* Zeitueberwachung rücksetzen *)
      	IP_C2.C_ENABLE := TRUE; (* Verbindungsaufbau freigeben *)
    	IP_C2.R_OBSERVE := FALSE; (* Empfangsueberwachung *)
    	R_BUF2.SIZE := UINT#0;
    	step := 120;

    120:IF IP_C2.C_STATE > BYTE#127 THEN (* FTP Datenkanal aufgebaut *)
    		IF FTP_DOWNLOAD THEN (* File von FTP empfangen *)
    			IP_C2.MAILBOX[3] := BYTE#1; (* IP Empfang sperren *)
    			step := 400;
    		ELSE
    			snd_text := 'STOR ';
    			next_step := 140;
    			snd_text := CONCAT(snd_text, ftp_path); (* STORE /PFAD/FILENAME *)
    			step := 999; (* Warten auf next_step *)
    		END_IF
    	END_IF

    (* ============== File an FTP senden ================ *)

    140:IF rcv_state = 125 OR rcv_state = 150 THEN (* 125 = Data connection already open / 150 = File status okay; about to open data connection *)
    		step := 160;
    	END_IF

    160:FSD.FILENAME := FILENAME; (* Dateiname *)
    	FSD.MODE := BYTE#1; (* vorhandene Datei zum lesen öffnen *)
    	FSD.OFFSET := UDINT#0; (* Start bei Dateianfang *)
    	S_BUF2.SIZE := UINT#65535; (* maximale länge einlesen *)
    	IP_C2.MAILBOX[2] := BYTE#1; (* IP Senden blockieren *)
    	step := 200;

    200:IF FSD.MODE = BYTE#0 AND FSD.ERROR = BYTE#0 THEN
    		IP_C2.MAILBOX[2] := BYTE#0; (* IP Senden erlauben *)
    		step := 210;
    	END_IF

    210:IF S_BUF2.SIZE = UINT#0 THEN (* warten bis alle daten gesendet sind *)
    		IF FSD.FILE_SIZE - FSD.OFFSET > UDINT#0 THEN
    			FSD.MODE := BYTE#1; (* vorhandene Datei zum lesen öffnen *)
    			S_BUF2.SIZE := UINT#65535; (* maximale länge einlesen *)
    			IP_C2.MAILBOX[2] := BYTE#1; (* IP Senden blockieren *)
    			step := 200;
    		ELSE
    			IP_C2.C_ENABLE := FALSE; (* FTP Datenkanal schliessen *)
    			step := 300;
    		END_IF
    	END_IF

    300:IF rcv_state = 226 THEN (* 226 Closing data connection. Requested file action successful  *)
    		snd_text := 'QUIT';
    		ip_c1_red_disable := TRUE;
    		next_step := 320;
    	END_IF

    320:IF rcv_state = 221 OR TON_WAIT.ET > timeout3  THEN (* 221 Service closing control connection *)
    		IP_C1.C_ENABLE := FALSE; (* FTP Steuerkanal schliessen *)
    		IF FILE_DELETE THEN (* Datei nach transfer löschen *)
    			FSD.MODE := BYTE#4; (* File Remove *)
    			step := 340;
    		ELSE
    			step := 900;
    		END_IF
    	END_IF

    340:IF FSD.MODE = BYTE#0 AND FSD.ERROR = BYTE#0 THEN
    		step := 900;
    	END_IF

    (*  ============== File vom FTP Empfangen  ============== *)

    400:snd_text := 'RETR ';
    	next_step := 410;
    	snd_text := CONCAT(snd_text, ftp_path); (* RETR /PFAD/FILENAME *)
    	step := 999; (* Warten auf next_step *)

    410:IF rcv_state = 125 OR rcv_state = 150 THEN (* 125 = Data connection already open / 150 = File status okay; about to open data connection *)
    		IP_C2.R_OBSERVE := TRUE; (* Empfangsueberwachung *)
    		step := 420;
    	END_IF

    420:FSD.FILENAME := FILENAME; (* Dateiname *)
    	FSD.MODE := BYTE#3; (* Datei neu anlegen *)
    	FSD.OFFSET := UDINT#0; (* Start bei Dateianfang *)
    	step := 460;

    440:IF R_BUF2.SIZE > UINT#0 THEN (* warten bis daten empfangen wurden *)
    		IP_C2.MAILBOX[3] := BYTE#1; (* IP Empfang blockieren bis Daten in Datei geschrieben wurden *)
    		FSD.MODE := BYTE#3; (* Daten in Datei schreiben *)
    		step := 460;
    	ELSIF FSD.FILE_SIZE = ftp_file_size THEN (* Verbindung abgebaut ? , oder 226 = Closing data connection. Requested file action successful *)
    		IP_C2.C_ENABLE := FALSE; (* FTP Datenkanal schliessen *)
    		ip_c2_red_disable := TRUE;
    		step := 700;
    	END_IF

    460:IF FSD.MODE = BYTE#0 AND FSD.ERROR = BYTE#0 THEN (* warten bis Daten geschreiben wurden *)
    		R_BUF2.SIZE := UINT#0; (* Daten löschen *)
    		IP_C2.MAILBOX[3] := BYTE#0; (* IP Empfang wieder erlauben *)
    		step := 440;
    	END_IF

    (* ================================================== *)

    700:IF rcv_state = 226 OR  TON_WAIT.ET > timeout3 THEN (* 226 Closing control connection. Requested file action successful  *)
    		IF FTP_DOWNLOAD AND FILE_DELETE THEN (* FTP Download und File löschen ? *)
    			snd_text := CONCAT('DELE ', ftp_path); (* DELE /PFAD/FILENAME *)
    			next_step := 720;
    		ELSE
    			step := 740;
    		END_IF
    	END_IF

    720:IF rcv_state = 250 THEN (* 250 Requested file action okay, completed *)
    		step := 740;
    	END_IF

    740:snd_text := 'QUIT';
    	ip_c1_red_disable := TRUE;
    	next_step := 760;
    	step := 999; (* Warten auf next_step *)

    760:IF rcv_state = 221 OR TON_WAIT.ET > timeout3 THEN (* 221 Service closing control connection  *)
    		IP_C1.C_ENABLE := FALSE; (* FTP Steuerkanal schliessen *)
    		IF NOT FTP_DOWNLOAD AND FILE_DELETE THEN (* FTP Upload und Datei nach transfer löschen *)
    			FSD.MODE := BYTE#4; (* File Remove *)
    			step := 780;
    		ELSE
    			step := 900;
    		END_IF
    	END_IF

    780:IF FSD.MODE = BYTE#0 AND FSD.ERROR = BYTE#0 THEN
    		step := 900;
    	END_IF

    (* ================================================== *)

    900:DONE := TRUE;
    	step := 980;

    980:IP_C1.C_ENABLE := FALSE; (* FTP Steuerkanal schliessen *)
    	IP_C2.C_ENABLE := FALSE; (* FTP Datenkanal schliessen *)
    	IP_C2.MAILBOX[2] := BYTE#0; (* IP Senden wieder erlauben *)
    	IP_C2.MAILBOX[3] := BYTE#0; (* IP Empfang wieder erlauben *)
    	S_BUF1.SIZE := UINT#0;
    	S_BUF2.SIZE := UINT#0;
    	R_BUF1.SIZE := UINT#0;
    	R_BUF2.SIZE := UINT#0;
    	ftp_file_size := UDINT#0;
    	snd_step := 0;
    	next_step := 0;
    	FSD.MODE := BYTE#5; (* Datei schliessen *)
    	step := 990;

    990:IF IP_C1.C_STATE = BYTE#0 AND IP_C2.C_STATE = BYTE#0 AND FSD.FILE_OPEN = FALSE THEN
    		step := 0;
    	END_IF

    999: ; (* Dummy Schritt, warten bis neuer schritt durch "next_step" aktiv wird *)

    END_CASE

    (* ++++++++++++++++++++++++++++++++++++++++++++++++++++++++++ *)

    IF step >= 30 THEN
    	IF R_BUF1.SIZE > UINT#0 THEN (* Daten wurden empfangen ? *)
    		idx1 := UINT_TO_INT(R_BUF1.SIZE);
    		REPEAT (* zeilenterminierung erkennen und echtes TEXT-Ende bestimmen *)
    			idx1 := idx1 - 1;
    		UNTIL idx1 = 0 OR R_BUF1.BUFFER[idx1] >= BYTE#32 (* TRUE = EXIT *)
    		END_REPEAT
    		idx1 := idx1 + 1; (* index auf SIZE umrechnen *)
    		rcv_text := BUFFER_TO_STRING(PT:=ADR(R_BUF1.BUFFER),SIZE:=idx1,START:=0,STOP:=STRING_LENGTH-1);
    		IF LEN(rcv_text) >= 3 THEN (* Statuscode prüfen und auswerten *)
    			str1 := LEFT(rcv_text,3);
    			IF IS_NUM(STR:=str1) THEN (* enthält nur Zahlen ? *)
    				rcv_state := STRING_TO_INT(str1);
    			END_IF
    			IP_C1.R_OBSERVE := FALSE;
    		END_IF
    		R_BUF1.SIZE := UINT#0; (* daten löschen *)

    	        (*####################  DEBUG-MESSAGE  ###################################*)
    	        (*IF _debug_enable THEN
    	          LOG_CL.NEW_MSG := 'RCV: >~1<';
    	          LOG_CL.PRINTF[1] := rcv_text;
    	          LOG_MSG();
    	        END_IF*)
    	        (*########################################################################*)

    	END_IF
    END_IF

    (* automatisches Datensenden *)

    CASE snd_step OF

    00:	IF LEN(snd_text) > 0 THEN
    	        (*####################  DEBUG-MESSAGE  ###################################*)
    	        (*IF _debug_enable THEN
    	          LOG_CL.NEW_MSG := 'SND: >~1<';
    	          LOG_CL.PRINTF[1] := snd_text;
    	          LOG_MSG();
    	        END_IF*)
    	        (*########################################################################*)
    		_STRING_TO_BUFFER(str:=snd_text,pos:=0,pt:=ADR(S_BUF1.BUFFER),size:=SIZEOF(S_BUF1.BUFFER)); (* String in puffer kopieren *)
    		idx1 := LEN(snd_text);
    		S_BUF1.BUFFER[idx1] := BYTE#16#0D;
    		idx1 := idx1 + 1;
    		S_BUF1.BUFFER[idx1] := BYTE#16#0A;
    		idx1 := idx1 + 1;
    		S_BUF1.SIZE := INT_TO_UINT(idx1); (* Sendelänge eintragen *)
    		R_BUF1.SIZE := UINT#0; (* Empfangsbuffer rücksetzen *)
    		IP_C1.R_OBSERVE := TRUE;
    		rcv_state := 9999; (* letzen FTP Status löschen *)
    		snd_text := '';
    		snd_step := 10;
    	END_IF

    10:	IF S_BUF1.SIZE = UINT#0 THEN (* warten bis alle daten gesendet sind *)
    		step := next_step;
    		snd_step := 0;
    	END_IF

    END_CASE

    (* Globale Fehlerbehandlung für Haupt-Routine *)
    IF ERROR_T = BYTE#0 AND step > 20 THEN (* noch kein Fehler gespeichert und Hauptroutine aktiv *)

    	IF IP_C1.ERROR > DWORD#0 AND IP_C1.C_ENABLE AND NOT IP_C1.TIME_RESET THEN  (* IP Control 1 *)
    		IF ip_c1_red_disable = FALSE OR IP_C1.ERROR <> DWORD#16#FD000000 THEN
    			ERROR_C := IP_C1.ERROR;
    			ERROR_T := BYTE#2;
    			step := 980;
    		END_IF
    	END_IF

    	IF IP_C2.ERROR > DWORD#0 AND IP_C2.C_ENABLE AND NOT IP_C2.TIME_RESET THEN  (* IP Control 2 *)
    		IF ip_c2_red_disable = FALSE OR IP_C2.ERROR <> DWORD#16#FD000000 THEN
    			ERROR_C := IP_C2.ERROR;
    			ERROR_T := BYTE#3;
    			step := 980;
    		END_IF
    	END_IF

    	IF FSD.MODE = BYTE#0 THEN
    		IF FSD.ERROR > BYTE#0 THEN
    			ERROR_C := BYTE_TO_DWORD(FSD.ERROR);
    			ERROR_T := BYTE#4; (* Dateizugriff *)
    			step := 980;
    		END_IF
    	END_IF
    END_IF

    IF TON_WAIT.Q THEN (* Ablaufstörung - Schrittkette *)
    	ERROR_C := SHL(INT_TO_DWORD(step),16) OR INT_TO_DWORD(rcv_state); (* aktuellen Schritt und letzten FTP Status eintragen *)
    	ERROR_T := BYTE#5;
    	step := 980;
    END_IF

    (* ######################################################## *)

    DNS_CLIENT(IP_C:=IP_C1, S_BUF:=S_BUF1, R_BUF:=R_BUF1, DOMAIN:=URL_DATA.DOMAIN, IP4_DNS:= DNS_IP4, ACTIVATE:=step=10); (* DNS-Client *)
    IPC1(IP:= DWORD#0, PORT:= WORD#0 , TIME_OUT:= TIMEOUT, IP_C:= IP_C1, S_BUF:= S_BUF1, R_BUF:= R_BUF1); (* FTP Steuerkanal *)
    IPC2(IP:= DWORD#0, PORT:= WORD#0 , TIME_OUT:= TIMEOUT, IP_C:= IP_C2, S_BUF:= S_BUF2, R_BUF:= R_BUF2); (* FTP Datenkanal *)

    TON_WAIT(IN:=step = last_step AND step > 0,PT:=timeout2);
    last_step := step;
    activate_last := ACTIVATE;
    BUSY := step <> 0;

    IF FTP_DOWNLOAD THEN (* FILE_SERVER *)
    	FS(FSD:=FSD,PT:=R_BUF2); (* Datei von FTP empfangen *)
    ELSE
    	FS(FSD:=FSD,PT:=S_BUF2); (* Datei an FTP senden *)
    END_IF

    (* revision history
    ks	05. may 2011	rev 1.3
    	FileServer AutoClose entfernt

    ks	11. may 2011	rev 1.2
    	ip_control - remote disconnect error ausblenden, und sonderbehandlung für pcworx

    ks	06. apr. 2011	rev 1.1
    	list_len und list_get durch element_count und element_get ersetzt

    ks	01. jan. 2011	rev 1.0
    	original version
    *)
END_FUNCTION_BLOCK

(* ---- GET_WAN_IP.st ---- *)
FUNCTION_BLOCK GET_WAN_IP
    (*http://www.oscat.de/images/OSCATNetwork/oscat_netlib121_en.pdf#page=96*)
    CASE state OF

    00:
    	IF ACTIVATE AND NOT activate_last THEN
    		state := 20;
    		DONE := FALSE;
    		ERROR_C := DWORD#0;
    		ERROR_T := BYTE#0;
    	END_IF

    20: (* URL for DNS UND HTTP-GET *)
    	URL_DATA := STRING_TO_URL(STR:='checkip.dyndns.com',DEFAULT_PROTOCOL:='',DEFAULT_PATH:='');
    	state := 40;

    40:
    	IF DNS_CLIENT.DONE THEN
    		state := 60;
    	ELSIF (DNS_CLIENT.ERROR > DWORD#00) THEN
    		(* Fehlerbehandlung *)
    		ERROR_C := DNS_CLIENT.ERROR;
    		ERROR_T := BYTE#01;
    		state := 100;
    	END_IF

    60:
    	IF HTTP_GET.DONE THEN
    		state := 80;
    	ELSIF (HTTP_GET.ERROR > DWORD#00) THEN
    		(* Fehlerbehandlung *)
    		ERROR_C := HTTP_GET.ERROR;
    		ERROR_T := BYTE#02;
    		state := 100;
    	END_IF

    80:
    	(* Als Antwort wird folgende HTML Seite empfangen , hier muss die IP-Adresse herauskopiert werden *)
    	(* <html><head><title>Current IP Check</title></head><body>Current IP Address: 85.127.217.33</body></html> *)
    	st_ip := '';
    	p1 := 0;
    	FOR i1 := UINT_TO_INT(HTTP_GET.BODY_START) TO UINT_TO_INT(HTTP_GET.BODY_STOP) DO
    		IF R_BUF.BUFFER[i1] = BYTE#58 THEN (* suche ':' *)
    			p1 := i1 + 2;
    			EXIT;
    		END_IF
    	END_FOR

    	p3 := p1 + 15;
    	IF p1 > 0 AND p3 < UINT_TO_INT(HTTP_GET.BODY_STOP) THEN
    		FOR p2 := p1 TO p3 DO
    			IF R_BUF.BUFFER[p2] <> BYTE#60 THEN (* suche '<' *)
    				st_ip := CONCAT(st_ip,CHR_TO_STRING(C:=R_BUF.BUFFER[p2]));
    			ELSE
    				EXIT;
    			END_IF
    		END_FOR
    	END_IF

    	WAN_IP4 := IP4_DECODE(STR:=st_ip);

    	IF WAN_IP4 <> DWORD#0 THEN
    		DONE := TRUE;
    		NEW_IP4 := WAN_IP4 <> wan_ip4_last;
    		wan_ip4_last := WAN_IP4;
    	ELSE
    		ERROR_C := DWORD#01; (* keine gültige IP gefunden *)
    		ERROR_T := BYTE#03;
    	END_IF
    	state := 100;

    100:
    	(* UNLOCK HTTP DATA *)
    	IF (NOT HTTP_GET.DONE) THEN
    		state := 0;
    		DONE := ERROR_T = BYTE#0;
    	END_IF

    END_CASE

    (* ---------------- DNS --------------- *)
    DNS_CLIENT(	IP_C:=IP_C,
    			S_BUF:=S_BUF,
    			R_BUF:=R_BUF,
    			DOMAIN:=URL_DATA.DOMAIN,
    			IP4_DNS:=DWORD#00,
    			ACTIVATE:=state=40 (* DNS Start *)
    			);
    (* nicht oder nicht direkt verwendete Parameter *)
    (* DWORD :=DNS_CLIENT.IP4;
       BOOL  :=DNS_CLIENT.DONE;
       BYTE  :=DNS_CLIENT.ERROR; *)
    (* -------------------------------------*)

    (* ------------- HTTP_GET --------------- *)

    HTTP_GET(	IP_C:=IP_C,
    			S_BUF:=S_BUF,
    			R_BUF:=R_BUF,
    			IP4:=DNS_CLIENT.IP4,
    			GET:=state=60,
    			MODE:=BYTE#2, (* HTTP 1.1 mit persistenter Verbindung *)
    			UNLOCK_BUF:=state=100,
    			URL_DATA:=URL_DATA
    			);

    (* nicht oder nicht direkt verwendete Parameter *)
    (*STRING := HTTP_GET.HTTP_STATUS;
      UINT :=HTTP_GET.HEADER_START;
      UINT :=HTTP_GET.HEADER_STOP;
      UINT :=HTTP_GET.BODY_START;
      UINT :=HTTP_GET.BODY_STOP;
      BOOL :=HTTP_GET.DONE;
      BYTE :=HTTP_GET.ERROR;
    *)
    (* -------------------------------------*)

    activate_last := ACTIVATE;

    (* revision history
    ks	28. dec 2009	rev 1.1
    	original version

    *)
END_FUNCTION_BLOCK
